LIN {X 0,Y 516.808,Z 520.516,A -85,B 0,C 180,E1 -4959.787,E2 -4959.787} C_VEL
LIN {X 0,Y 517.098,Z 512.267,A -85,B 0,C 180,E1 -4960.969,E2 -4960.969} C_VEL
LIN {X 0,Y 517.442,Z 502.246,A -85,B 0,C 180,E1 -4962.162,E2 -4962.162} C_VEL
LIN {X 0,Y 517.823,Z 491.268,A -85,B 0,C 180,E1 -4963.24,E2 -4963.24} C_VEL
LIN {X 0,Y 518.232,Z 480.256,A -85,B 0,C 180,E1 -4964.129,E2 -4964.129} C_VEL
LIN {X 0,Y 518.655,Z 468.311,A -85,B 0,C 180,E1 -4964.919,E2 -4964.919} C_VEL
LIN {X 0,Y 519.002,Z 455.123,A -85,B 0,C 180,E1 -4965.613,E2 -4965.613} C_VEL
LIN {X 0,Y 519.331,Z 440.839,A -85,B 0,C 180,E1 -4966.176,E2 -4966.176} C_VEL
LIN {X 0,Y 519.289,Z 432.051,A -85,B 0,C 180,E1 -4966.444,E2 -4966.444} C_VEL
LIN {X 0,Y 516.421,Z 418.731,A -85,B 0,C 180,E1 -4966.835,E2 -4966.835} C_VEL
LIN {X 0,Y 516.476,Z 412.491,A -85,B 0,C 180,E1 -4970.128,E2 -4970.128} C_VEL
LIN {X 0,Y 516.541,Z 406.65,A -85,B 0,C 180,E1 -4973.239,E2 -4973.239} C_VEL
LIN {X 0,Y 516.631,Z 401.356,A -85,B 0,C 180,E1 -4976.125,E2 -4976.125} C_VEL
LIN {X 0,Y 516.771,Z 395.647,A -85,B 0,C 180,E1 -4979.314,E2 -4979.314} C_VEL
LIN {X 0,Y 516.843,Z 390.925,A -85,B 0,C 180,E1 -4982.027,E2 -4982.027} C_VEL
LIN {X 0,Y 516.93,Z 386.203,A -85,B 0,C 180,E1 -4984.821,E2 -4984.821} C_VEL
LIN {X 0,Y 517.027,Z 381.474,A -85,B 0,C 180,E1 -4987.712,E2 -4987.712} C_VEL
LIN {X 0,Y 516.923,Z 379.126,A -85,B 0,C 180,E1 -4989.198,E2 -4989.198} C_VEL
LIN {X 0,Y 516.879,Z 378.732,A -85,B 0,C 180,E1 -4989.722,E2 -4989.722} C_VEL
LIN {X 0,Y 516.909,Z 378.724,A -85,B 0,C 180,E1 -4992.761,E2 -4992.761} C_VEL
LIN {X 0,Y 516.926,Z 378.721,A -85,B 0,C 180,E1 -4995.01,E2 -4995.01} C_VEL
LIN {X 0,Y 516.918,Z 378.721,A -85,B 0,C 180,E1 -4998.399,E2 -4998.399} C_VEL
LIN {X 0,Y 516.884,Z 378.727,A -85,B 0,C 180,E1 -5001.284,E2 -5001.284} C_VEL
LIN {X 0,Y 516.894,Z 378.726,A -85,B 0,C 180,E1 -5004.221,E2 -5004.221} C_VEL
LIN {X 0,Y 516.898,Z 378.722,A -85,B 0,C 180,E1 -5007.053,E2 -5007.053} C_VEL
LIN {X 0,Y 516.895,Z 378.722,A -85,B 0,C 180,E1 -5009.796,E2 -5009.796} C_VEL
LIN {X 0,Y 516.931,Z 378.723,A -85,B 0,C 180,E1 -5012.467,E2 -5012.467} C_VEL
LIN {X 0,Y 516.912,Z 378.72,A -85,B 0,C 180,E1 -5015.072,E2 -5015.072} C_VEL
LIN {X 0,Y 516.889,Z 378.723,A -85,B 0,C 180,E1 -5018.462,E2 -5018.462} C_VEL
LIN {X 0,Y 516.905,Z 378.722,A -85,B 0,C 180,E1 -5020.955,E2 -5020.955} C_VEL
LIN {X 0,Y 516.917,Z 378.72,A -85,B 0,C 180,E1 -5023.41,E2 -5023.41} C_VEL
LIN {X 0,Y 516.909,Z 378.721,A -85,B 0,C 180,E1 -5025.834,E2 -5025.834} C_VEL
LIN {X 0,Y 516.954,Z 378.716,A -85,B 0,C 180,E1 -5029.028,E2 -5029.028} C_VEL
LIN {X 0,Y 516.982,Z 378.714,A -85,B 0,C 180,E1 -5032.187,E2 -5032.187} C_VEL
LIN {X 0,Y 517.033,Z 378.704,A -85,B 0,C 180,E1 -5034.54,E2 -5034.54} C_VEL
LIN {X 0,Y 517.086,Z 378.698,A -85,B 0,C 180,E1 -5037.663,E2 -5037.663} C_VEL
LIN {X 0,Y 517.097,Z 378.696,A -85,B 0,C 180,E1 -5040.779,E2 -5040.779} C_VEL
LIN {X 0,Y 517.017,Z 378.71,A -85,B 0,C 180,E1 -5043.117,E2 -5043.117} C_VEL
LIN {X 0,Y 517.013,Z 378.709,A -85,B 0,C 180,E1 -5046.243,E2 -5046.243} C_VEL
LIN {X 0,Y 516.953,Z 378.716,A -85,B 0,C 180,E1 -5049.389,E2 -5049.389} C_VEL
LIN {X 0,Y 516.956,Z 378.715,A -85,B 0,C 180,E1 -5051.807,E2 -5051.807} C_VEL
LIN {X 0,Y 516.951,Z 378.715,A -85,B 0,C 180,E1 -5055.148,E2 -5055.148} C_VEL
LIN {X 0,Y 516.929,Z 378.719,A -85,B 0,C 180,E1 -5058.222,E2 -5058.222} C_VEL
LIN {X 0,Y 516.916,Z 378.721,A -85,B 0,C 180,E1 -5060.701,E2 -5060.701} C_VEL
LIN {X 0,Y 516.915,Z 378.72,A -85,B 0,C 180,E1 -5064.072,E2 -5064.072} C_VEL
LIN {X 0,Y 516.928,Z 378.717,A -85,B 0,C 180,E1 -5066.658,E2 -5066.658} C_VEL
LIN {X 0,Y 516.914,Z 378.72,A -85,B 0,C 180,E1 -5069.524,E2 -5069.524} C_VEL
LIN {X 0,Y 516.898,Z 378.727,A -85,B 0,C 180,E1 -5072.543,E2 -5072.543} C_VEL
LIN {X 0,Y 516.886,Z 378.725,A -85,B 0,C 180,E1 -5075.332,E2 -5075.332} C_VEL
LIN {X 0,Y 516.884,Z 378.725,A -85,B 0,C 180,E1 -5077.943,E2 -5077.943} C_VEL
LIN {X 0,Y 516.907,Z 378.725,A -85,B 0,C 180,E1 -5080.74,E2 -5080.74} C_VEL
LIN {X 0,Y 516.884,Z 378.729,A -85,B 0,C 180,E1 -5083.903,E2 -5083.903} C_VEL
LIN {X 0,Y 516.887,Z 378.729,A -85,B 0,C 180,E1 -5087.169,E2 -5087.169} C_VEL
LIN {X 0,Y 516.955,Z 378.759,A -85,B 0,C 180,E1 -5089.779,E2 -5089.779} C_VEL
LIN {X 0,Y 517.287,Z 382.793,A -85,B 0,C 180,E1 -5091.999,E2 -5091.999} C_VEL
LIN {X 0,Y 517.184,Z 387.817,A -85,B 0,C 180,E1 -5094.621,E2 -5094.621} C_VEL
LIN {X 0,Y 517.022,Z 393.407,A -85,B 0,C 180,E1 -5097.435,E2 -5097.435} C_VEL
LIN {X 0,Y 516.898,Z 399.648,A -85,B 0,C 180,E1 -5100.479,E2 -5100.479} C_VEL
LIN {X 0,Y 516.724,Z 405.675,A -85,B 0,C 180,E1 -5103.331,E2 -5103.331} C_VEL
LIN {X 0,Y 516.658,Z 411.289,A -85,B 0,C 180,E1 -5105.915,E2 -5105.915} C_VEL
LIN {X 0,Y 516.578,Z 416.905,A -85,B 0,C 180,E1 -5108.449,E2 -5108.449} C_VEL
LIN {X 0,Y 516.49,Z 422.509,A -85,B 0,C 180,E1 -5110.939,E2 -5110.939} C_VEL
LIN {X 0,Y 516.463,Z 427.639,A -85,B 0,C 180,E1 -5113.192,E2 -5113.192} C_VEL
LIN {X 0,Y 519.514,Z 442.817,A -85,B 0,C 180,E1 -5113.639,E2 -5113.639} C_VEL
LIN {X 0,Y 519.207,Z 456.026,A -85,B 0,C 180,E1 -5114.065,E2 -5114.065} C_VEL
LIN {X 0,Y 518.82,Z 469.992,A -85,B 0,C 180,E1 -5114.683,E2 -5114.683} C_VEL
LIN {X 0,Y 518.478,Z 482.084,A -85,B 0,C 180,E1 -5115.377,E2 -5115.377} C_VEL
LIN {X 0,Y 518.093,Z 493.307,A -85,B 0,C 180,E1 -5116.167,E2 -5116.167} C_VEL
LIN {X 0,Y 517.657,Z 504.851,A -85,B 0,C 180,E1 -5117.155,E2 -5117.155} C_VEL
LIN {X 0,Y 517.334,Z 515.308,A -85,B 0,C 180,E1 -5118.242,E2 -5118.242} C_VEL
LIN {X 0,Y 517.002,Z 524.755,A -85,B 0,C 180,E1 -5119.425,E2 -5119.425} C_VEL
LIN {X 0,Y 516.71,Z 533.754,A -85,B 0,C 180,E1 -5120.804,E2 -5120.804} C_VEL
LIN {X 0,Y 516.501,Z 541.022,A -85,B 0,C 180,E1 -5122.179,E2 -5122.179} C_VEL
LIN {X 0,Y 516.396,Z 547.553,A -85,B 0,C 180,E1 -5123.749,E2 -5123.749} C_VEL
LIN {X 0,Y 516.306,Z 551.373,A -85,B 0,C 180,E1 -5124.924,E2 -5124.924} C_VEL
LIN {X 0,Y 516.325,Z 554.315,A -85,B 0,C 180,E1 -5126.097,E2 -5126.097} C_VEL
LIN {X 0,Y 516.26,Z 557.002,A -85,B 0,C 180,E1 -5127.659,E2 -5127.659} C_VEL
LIN {X 0,Y 516.157,Z 558.334,A -85,B 0,C 180,E1 -5129.22,E2 -5129.22} C_VEL
LIN {X 0,Y 516.157,Z 558.334,A -85,B 0,C 180,E1 -5130.78,E2 -5130.78} C_VEL
LIN {X 0,Y 516.259,Z 557.005,A -85,B 0,C 180,E1 -5132.341,E2 -5132.341} C_VEL
LIN {X 0,Y 516.325,Z 554.32,A -85,B 0,C 180,E1 -5133.902,E2 -5133.902} C_VEL
LIN {X 0,Y 516.388,Z 550.192,A -85,B 0,C 180,E1 -5135.467,E2 -5135.467} C_VEL
LIN {X 0,Y 516.405,Z 544.503,A -85,B 0,C 180,E1 -5137.035,E2 -5137.035} C_VEL
LIN {X 0,Y 516.599,Z 538.089,A -85,B 0,C 180,E1 -5138.409,E2 -5138.409} C_VEL
LIN {X 0,Y 516.827,Z 530.119,A -85,B 0,C 180,E1 -5139.787,E2 -5139.787} C_VEL
LIN {X 0,Y 517.109,Z 521.781,A -85,B 0,C 180,E1 -5140.969,E2 -5140.969} C_VEL
LIN {X 0,Y 517.458,Z 511.344,A -85,B 0,C 180,E1 -5142.197,E2 -5142.197} C_VEL
LIN {X 0,Y 517.812,Z 500.543,A -85,B 0,C 180,E1 -5143.24,E2 -5143.24} C_VEL
LIN {X 0,Y 518.256,Z 487.977,A -85,B 0,C 180,E1 -5144.229,E2 -5144.229} C_VEL
LIN {X 0,Y 518.701,Z 475.501,A -85,B 0,C 180,E1 -5145.018,E2 -5145.018} C_VEL
LIN {X 0,Y 519.038,Z 462.675,A -85,B 0,C 180,E1 -5145.662,E2 -5145.662} C_VEL
LIN {X 0,Y 519.367,Z 449.107,A -85,B 0,C 180,E1 -5146.176,E2 -5146.176} C_VEL
LIN {X 0,Y 519.32,Z 441.383,A -85,B 0,C 180,E1 -5146.407,E2 -5146.407} C_VEL
LIN {X 0,Y 516.463,Z 427.607,A -85,B 0,C 180,E1 -5146.808,E2 -5146.808} C_VEL
LIN {X 0,Y 516.572,Z 419.95,A -85,B 0,C 180,E1 -5150.157,E2 -5150.157} C_VEL
LIN {X 0,Y 516.615,Z 413.124,A -85,B 0,C 180,E1 -5153.236,E2 -5153.236} C_VEL
LIN {X 0,Y 516.725,Z 406.793,A -85,B 0,C 180,E1 -5156.147,E2 -5156.147} C_VEL
LIN {X 0,Y 516.814,Z 401.952,A -85,B 0,C 180,E1 -5158.421,E2 -5158.421} C_VEL
LIN {X 0,Y 516.969,Z 396.377,A -85,B 0,C 180,E1 -5161.104,E2 -5161.104} C_VEL
LIN {X 0,Y 517.109,Z 390.531,A -85,B 0,C 180,E1 -5163.999,E2 -5163.999} C_VEL
LIN {X 0,Y 517.263,Z 385.229,A -85,B 0,C 180,E1 -5166.714,E2 -5166.714} C_VEL
LIN {X 0,Y 517.184,Z 380.519,A -85,B 0,C 180,E1 -5169.234,E2 -5169.234} C_VEL
LIN {X 0,Y 516.936,Z 378.724,A -85,B 0,C 180,E1 -5170.351,E2 -5170.351} C_VEL
LIN {X 0,Y 516.886,Z 378.728,A -85,B 0,C 180,E1 -5172.831,E2 -5172.831} C_VEL
LIN {X 0,Y 516.883,Z 378.729,A -85,B 0,C 180,E1 -5176.097,E2 -5176.097} C_VEL
LIN {X 0,Y 516.906,Z 378.725,A -85,B 0,C 180,E1 -5179.26,E2 -5179.26} C_VEL
LIN {X 0,Y 516.887,Z 378.723,A -85,B 0,C 180,E1 -5182.056,E2 -5182.056} C_VEL
LIN {X 0,Y 516.897,Z 378.722,A -85,B 0,C 180,E1 -5185.176,E2 -5185.176} C_VEL
LIN {X 0,Y 516.878,Z 378.726,A -85,B 0,C 180,E1 -5187.975,E2 -5187.975} C_VEL
LIN {X 0,Y 516.923,Z 378.723,A -85,B 0,C 180,E1 -5190.696,E2 -5190.696} C_VEL
LIN {X 0,Y 516.944,Z 378.719,A -85,B 0,C 180,E1 -5193.804,E2 -5193.804} C_VEL
LIN {X 0,Y 516.867,Z 378.726,A -85,B 0,C 180,E1 -5196.776,E2 -5196.776} C_VEL
LIN {X 0,Y 516.941,Z 378.716,A -85,B 0,C 180,E1 -5199.732,E2 -5199.732} C_VEL
LIN {X 0,Y 516.931,Z 378.718,A -85,B 0,C 180,E1 -5202.596,E2 -5202.596} C_VEL
LIN {X 0,Y 516.953,Z 378.716,A -85,B 0,C 180,E1 -5205.03,E2 -5205.03} C_VEL
LIN {X 0,Y 516.968,Z 378.714,A -85,B 0,C 180,E1 -5208.234,E2 -5208.234} C_VEL
LIN {X 0,Y 516.971,Z 378.713,A -85,B 0,C 180,E1 -5211.4,E2 -5211.4} C_VEL
LIN {X 0,Y 517.012,Z 378.71,A -85,B 0,C 180,E1 -5213.757,E2 -5213.757} C_VEL
LIN {X 0,Y 517.086,Z 378.698,A -85,B 0,C 180,E1 -5217.663,E2 -5217.663} C_VEL
LIN {X 0,Y 517.096,Z 378.696,A -85,B 0,C 180,E1 -5220.779,E2 -5220.779} C_VEL
LIN {X 0,Y 517.015,Z 378.711,A -85,B 0,C 180,E1 -5223.117,E2 -5223.117} C_VEL
LIN {X 0,Y 517.012,Z 378.71,A -85,B 0,C 180,E1 -5226.243,E2 -5226.243} C_VEL
LIN {X 0,Y 516.954,Z 378.716,A -85,B 0,C 180,E1 -5229.389,E2 -5229.389} C_VEL
LIN {X 0,Y 516.954,Z 378.715,A -85,B 0,C 180,E1 -5231.807,E2 -5231.807} C_VEL
LIN {X 0,Y 516.95,Z 378.715,A -85,B 0,C 180,E1 -5235.148,E2 -5235.148} C_VEL
LIN {X 0,Y 516.928,Z 378.719,A -85,B 0,C 180,E1 -5238.222,E2 -5238.222} C_VEL
LIN {X 0,Y 516.915,Z 378.721,A -85,B 0,C 180,E1 -5240.701,E2 -5240.701} C_VEL
LIN {X 0,Y 516.914,Z 378.722,A -85,B 0,C 180,E1 -5244.072,E2 -5244.072} C_VEL
LIN {X 0,Y 516.928,Z 378.717,A -85,B 0,C 180,E1 -5246.658,E2 -5246.658} C_VEL
LIN {X 0,Y 516.913,Z 378.721,A -85,B 0,C 180,E1 -5249.524,E2 -5249.524} C_VEL
LIN {X 0,Y 516.898,Z 378.726,A -85,B 0,C 180,E1 -5252.543,E2 -5252.543} C_VEL
LIN {X 0,Y 516.886,Z 378.725,A -85,B 0,C 180,E1 -5255.333,E2 -5255.333} C_VEL
LIN {X 0,Y 516.887,Z 378.722,A -85,B 0,C 180,E1 -5257.944,E2 -5257.944} C_VEL
LIN {X 0,Y 516.887,Z 378.727,A -85,B 0,C 180,E1 -5260.741,E2 -5260.741} C_VEL
LIN {X 0,Y 516.886,Z 378.724,A -85,B 0,C 180,E1 -5262.831,E2 -5262.831} C_VEL
LIN {X 0,Y 516.925,Z 378.72,A -85,B 0,C 180,E1 -5265.01,E2 -5265.01} C_VEL
LIN {X 0,Y 516.92,Z 378.722,A -85,B 0,C 180,E1 -5268.398,E2 -5268.398} C_VEL
LIN {X 0,Y 516.869,Z 378.743,A -85,B 0,C 180,E1 -5270.303,E2 -5270.303} C_VEL
LIN {X 0,Y 516.232,Z 379.398,A -85,B 0,C 180,E1 -5270.949,E2 -5270.949} C_VEL
LIN {X 0,Y 513.459,Z 381.35,A -85,B 0,C 180,E1 -5271.988,E2 -5271.988} C_VEL
LIN {X 0,Y 511.089,Z 383.022,A -85,B 0,C 180,E1 -5272.82,E2 -5272.82} C_VEL
LIN {X 0,Y 510.047,Z 384.192,A -85,B 0,C 180,E1 -5273.464,E2 -5273.464} C_VEL
LIN {X 0,Y 509.95,Z 384.556,A -85,B 0,C 180,E1 -5273.682,E2 -5273.682} C_VEL
LIN {X 0,Y 509.869,Z 389.232,A -85,B 0,C 180,E1 -5276.54,E2 -5276.54} C_VEL
LIN {X 0,Y 509.747,Z 393.955,A -85,B 0,C 180,E1 -5279.328,E2 -5279.328} C_VEL
LIN {X 0,Y 509.631,Z 398.68,A -85,B 0,C 180,E1 -5282.039,E2 -5282.039} C_VEL
LIN {X 0,Y 509.537,Z 403.392,A -85,B 0,C 180,E1 -5284.686,E2 -5284.686} C_VEL
LIN {X 0,Y 509.476,Z 408.613,A -85,B 0,C 180,E1 -5287.554,E2 -5287.554} C_VEL
LIN {X 0,Y 509.339,Z 414.363,A -85,B 0,C 180,E1 -5290.661,E2 -5290.661} C_VEL
LIN {X 0,Y 509.343,Z 418.805,A -85,B 0,C 180,E1 -5293.027,E2 -5293.027} C_VEL
LIN {X 0,Y 512.636,Z 433.906,A -85,B 0,C 180,E1 -5293.477,E2 -5293.477} C_VEL
LIN {X 0,Y 512.426,Z 446.731,A -85,B 0,C 180,E1 -5293.907,E2 -5293.907} C_VEL
LIN {X 0,Y 512.057,Z 459.474,A -85,B 0,C 180,E1 -5294.476,E2 -5294.476} C_VEL
LIN {X 0,Y 511.653,Z 471.727,A -85,B 0,C 180,E1 -5295.177,E2 -5295.177} C_VEL
LIN {X 0,Y 511.216,Z 483.048,A -85,B 0,C 180,E1 -5295.978,E2 -5295.978} C_VEL
LIN {X 0,Y 510.749,Z 494.653,A -85,B 0,C 180,E1 -5296.978,E2 -5296.978} C_VEL
LIN {X 0,Y 510.302,Z 505.157,A -85,B 0,C 180,E1 -5298.078,E2 -5298.078} C_VEL
LIN {X 0,Y 510.018,Z 514.633,A -85,B 0,C 180,E1 -5299.279,E2 -5299.279} C_VEL
LIN {X 0,Y 509.69,Z 523.679,A -85,B 0,C 180,E1 -5300.676,E2 -5300.676} C_VEL
LIN {X 0,Y 509.457,Z 530.96,A -85,B 0,C 180,E1 -5302.071,E2 -5302.071} C_VEL
LIN {X 0,Y 509.308,Z 537.501,A -85,B 0,C 180,E1 -5303.662,E2 -5303.662} C_VEL
LIN {X 0,Y 509.239,Z 541.346,A -85,B 0,C 180,E1 -5304.853,E2 -5304.853} C_VEL
LIN {X 0,Y 509.235,Z 544.295,A -85,B 0,C 180,E1 -5306.043,E2 -5306.043} C_VEL
LIN {X 0,Y 509.189,Z 547.011,A -85,B 0,C 180,E1 -5307.627,E2 -5307.627} C_VEL
LIN {X 0,Y 509.07,Z 548.377,A -85,B 0,C 180,E1 -5309.209,E2 -5309.209} C_VEL
LIN {X 0,Y 509.071,Z 548.419,A -85,B 0,C 180,E1 -5310.791,E2 -5310.791} C_VEL
LIN {X 0,Y 509.188,Z 547.134,A -85,B 0,C 180,E1 -5312.373,E2 -5312.373} C_VEL
LIN {X 0,Y 509.235,Z 544.493,A -85,B 0,C 180,E1 -5313.957,E2 -5313.957} C_VEL
LIN {X 0,Y 509.314,Z 540.427,A -85,B 0,C 180,E1 -5315.543,E2 -5315.543} C_VEL
LIN {X 0,Y 509.356,Z 534.811,A -85,B 0,C 180,E1 -5317.134,E2 -5317.134} C_VEL
LIN {X 0,Y 509.548,Z 528.468,A -85,B 0,C 180,E1 -5318.527,E2 -5318.527} C_VEL
LIN {X 0,Y 509.773,Z 520.582,A -85,B 0,C 180,E1 -5319.924,E2 -5319.924} C_VEL
LIN {X 0,Y 510.103,Z 512.332,A -85,B 0,C 180,E1 -5321.121,E2 -5321.121} C_VEL
LIN {X 0,Y 510.453,Z 502.664,A -85,B 0,C 180,E1 -5322.291,E2 -5322.291} C_VEL
LIN {X 0,Y 510.905,Z 491.33,A -85,B 0,C 180,E1 -5323.423,E2 -5323.423} C_VEL
LIN {X 0,Y 511.323,Z 480.317,A -85,B 0,C 180,E1 -5324.324,E2 -5324.324} C_VEL
LIN {X 0,Y 511.776,Z 468.369,A -85,B 0,C 180,E1 -5325.125,E2 -5325.125} C_VEL
LIN {X 0,Y 512.163,Z 455.177,A -85,B 0,C 180,E1 -5325.827,E2 -5325.827} C_VEL
LIN {X 0,Y 512.504,Z 441.427,A -85,B 0,C 180,E1 -5326.38,E2 -5326.38} C_VEL
LIN {X 0,Y 512.552,Z 433.522,A -85,B 0,C 180,E1 -5326.626,E2 -5326.626} C_VEL
LIN {X 0,Y 509.338,Z 418.801,A -85,B 0,C 180,E1 -5327.077,E2 -5327.077} C_VEL
LIN {X 0,Y 509.419,Z 412.833,A -85,B 0,C 180,E1 -5330.259,E2 -5330.259} C_VEL
LIN {X 0,Y 509.465,Z 408.266,A -85,B 0,C 180,E1 -5332.722,E2 -5332.722} C_VEL
LIN {X 0,Y 509.538,Z 403.554,A -85,B 0,C 180,E1 -5335.314,E2 -5335.314} C_VEL
LIN {X 0,Y 509.63,Z 398.693,A -85,B 0,C 180,E1 -5338.044,E2 -5338.044} C_VEL
LIN {X 0,Y 509.747,Z 394.111,A -85,B 0,C 180,E1 -5340.672,E2 -5340.672} C_VEL
LIN {X 0,Y 509.862,Z 389.385,A -85,B 0,C 180,E1 -5343.461,E2 -5343.461} C_VEL
LIN {X 0,Y 509.95,Z 384.66,A -85,B 0,C 180,E1 -5346.343,E2 -5346.343} C_VEL
LIN {X 0,Y 509.954,Z 381.496,A -85,B 0,C 180,E1 -5348.329,E2 -5348.329} C_VEL
LIN {X 0,Y 509.843,Z 379.737,A -85,B 0,C 180,E1 -5349.471,E2 -5349.471} C_VEL
LIN {X 0,Y 509.85,Z 379.601,A -85,B 0,C 180,E1 -5352.488,E2 -5352.488} C_VEL
LIN {X 0,Y 509.86,Z 379.599,A -85,B 0,C 180,E1 -5355.332,E2 -5355.332} C_VEL
LIN {X 0,Y 509.86,Z 379.6,A -85,B 0,C 180,E1 -5358.575,E2 -5358.575} C_VEL
LIN {X 0,Y 509.854,Z 379.599,A -85,B 0,C 180,E1 -5361.786,E2 -5361.786} C_VEL
LIN {X 0,Y 509.85,Z 379.602,A -85,B 0,C 180,E1 -5364.623,E2 -5364.623} C_VEL
LIN {X 0,Y 509.864,Z 379.602,A -85,B 0,C 180,E1 -5367.481,E2 -5367.481} C_VEL
LIN {X 0,Y 509.862,Z 379.598,A -85,B 0,C 180,E1 -5370.274,E2 -5370.274} C_VEL
LIN {X 0,Y 509.888,Z 379.596,A -85,B 0,C 180,E1 -5372.944,E2 -5372.944} C_VEL
LIN {X 0,Y 509.868,Z 379.601,A -85,B 0,C 180,E1 -5375.574,E2 -5375.574} C_VEL
LIN {X 0,Y 509.854,Z 379.602,A -85,B 0,C 180,E1 -5378.998,E2 -5378.998} C_VEL
LIN {X 0,Y 509.885,Z 379.598,A -85,B 0,C 180,E1 -5382.001,E2 -5382.001} C_VEL
LIN {X 0,Y 509.914,Z 379.591,A -85,B 0,C 180,E1 -5384.819,E2 -5384.819} C_VEL
LIN {X 0,Y 509.904,Z 379.593,A -85,B 0,C 180,E1 -5388.124,E2 -5388.124} C_VEL
LIN {X 0,Y 509.918,Z 379.59,A -85,B 0,C 180,E1 -5391.28,E2 -5391.28} C_VEL
LIN {X 0,Y 509.982,Z 379.587,A -85,B 0,C 180,E1 -5393.67,E2 -5393.67} C_VEL
LIN {X 0,Y 510.057,Z 379.573,A -85,B 0,C 180,E1 -5397.631,E2 -5397.631} C_VEL
LIN {X 0,Y 510.067,Z 379.571,A -85,B 0,C 180,E1 -5400.789,E2 -5400.789} C_VEL
LIN {X 0,Y 509.959,Z 379.59,A -85,B 0,C 180,E1 -5403.16,E2 -5403.16} C_VEL
LIN {X 0,Y 509.981,Z 379.586,A -85,B 0,C 180,E1 -5406.33,E2 -5406.33} C_VEL
LIN {X 0,Y 509.915,Z 379.591,A -85,B 0,C 180,E1 -5408.72,E2 -5408.72} C_VEL
LIN {X 0,Y 509.908,Z 379.592,A -85,B 0,C 180,E1 -5411.932,E2 -5411.932} C_VEL
LIN {X 0,Y 509.897,Z 379.594,A -85,B 0,C 180,E1 -5415.242,E2 -5415.242} C_VEL
LIN {X 0,Y 509.892,Z 379.598,A -85,B 0,C 180,E1 -5418.001,E2 -5418.001} C_VEL
LIN {X 0,Y 509.854,Z 379.604,A -85,B 0,C 180,E1 -5421.002,E2 -5421.002} C_VEL
LIN {X 0,Y 509.84,Z 379.599,A -85,B 0,C 180,E1 -5423.563,E2 -5423.563} C_VEL
LIN {X 0,Y 509.914,Z 379.592,A -85,B 0,C 180,E1 -5426.378,E2 -5426.378} C_VEL
LIN {X 0,Y 509.879,Z 379.597,A -85,B 0,C 180,E1 -5428.844,E2 -5428.844} C_VEL
LIN {X 0,Y 509.822,Z 379.603,A -85,B 0,C 180,E1 -5431.59,E2 -5431.59} C_VEL
LIN {X 0,Y 509.857,Z 379.601,A -85,B 0,C 180,E1 -5434.413,E2 -5434.413} C_VEL
LIN {X 0,Y 509.822,Z 379.61,A -85,B 0,C 180,E1 -5437.34,E2 -5437.34} C_VEL
LIN {X 0,Y 509.864,Z 379.603,A -85,B 0,C 180,E1 -5440.38,E2 -5440.38} C_VEL
LIN {X 0,Y 509.825,Z 379.604,A -85,B 0,C 180,E1 -5443.062,E2 -5443.062} C_VEL
LIN {X 0,Y 509.825,Z 379.606,A -85,B 0,C 180,E1 -5445.793,E2 -5445.793} C_VEL
LIN {X 0,Y 509.864,Z 379.603,A -85,B 0,C 180,E1 -5448.575,E2 -5448.575} C_VEL
LIN {X 0,Y 509.913,Z 379.659,A -85,B 0,C 180,E1 -5449.625,E2 -5449.625} C_VEL
LIN {X 0,Y 510.253,Z 383.408,A -85,B 0,C 180,E1 -5451.729,E2 -5451.729} C_VEL
LIN {X 0,Y 510.177,Z 388.375,A -85,B 0,C 180,E1 -5454.367,E2 -5454.367} C_VEL
LIN {X 0,Y 509.979,Z 394.483,A -85,B 0,C 180,E1 -5457.489,E2 -5457.489} C_VEL
LIN {X 0,Y 509.858,Z 400.107,A -85,B 0,C 180,E1 -5460.274,E2 -5460.274} C_VEL
LIN {X 0,Y 509.703,Z 405.632,A -85,B 0,C 180,E1 -5462.934,E2 -5462.934} C_VEL
LIN {X 0,Y 509.618,Z 411.219,A -85,B 0,C 180,E1 -5465.561,E2 -5465.561} C_VEL
LIN {X 0,Y 509.535,Z 416.831,A -85,B 0,C 180,E1 -5468.136,E2 -5468.136} C_VEL
LIN {X 0,Y 509.418,Z 422.437,A -85,B 0,C 180,E1 -5470.664,E2 -5470.664} C_VEL
LIN {X 0,Y 509.369,Z 427.567,A -85,B 0,C 180,E1 -5472.95,E2 -5472.95} C_VEL
LIN {X 0,Y 512.686,Z 443.983,A -85,B 0,C 180,E1 -5473.449,E2 -5473.449} C_VEL
LIN {X 0,Y 512.373,Z 456.977,A -85,B 0,C 180,E1 -5473.887,E2 -5473.887} C_VEL
LIN {X 0,Y 511.967,Z 469.923,A -85,B 0,C 180,E1 -5474.473,E2 -5474.473} C_VEL
LIN {X 0,Y 511.598,Z 482.015,A -85,B 0,C 180,E1 -5475.175,E2 -5475.175} C_VEL
LIN {X 0,Y 511.141,Z 493.238,A -85,B 0,C 180,E1 -5475.975,E2 -5475.975} C_VEL
LIN {X 0,Y 510.703,Z 504.781,A -85,B 0,C 180,E1 -5476.977,E2 -5476.977} C_VEL
LIN {X 0,Y 510.34,Z 515.239,A -85,B 0,C 180,E1 -5478.079,E2 -5478.079} C_VEL
LIN {X 0,Y 509.991,Z 524.686,A -85,B 0,C 180,E1 -5479.278,E2 -5479.278} C_VEL
LIN {X 0,Y 509.673,Z 533.685,A -85,B 0,C 180,E1 -5480.676,E2 -5480.676} C_VEL
LIN {X 0,Y 509.45,Z 540.953,A -85,B 0,C 180,E1 -5482.071,E2 -5482.071} C_VEL
LIN {X 0,Y 509.311,Z 547.484,A -85,B 0,C 180,E1 -5483.662,E2 -5483.662} C_VEL
LIN {X 0,Y 509.239,Z 551.304,A -85,B 0,C 180,E1 -5484.853,E2 -5484.853} C_VEL
LIN {X 0,Y 509.218,Z 554.248,A -85,B 0,C 180,E1 -5486.043,E2 -5486.043} C_VEL
LIN {X 0,Y 509.159,Z 556.942,A -85,B 0,C 180,E1 -5487.627,E2 -5487.627} C_VEL
LIN {X 0,Y 509.071,Z 558.276,A -85,B 0,C 180,E1 -5489.209,E2 -5489.209} C_VEL
LIN {X 0,Y 509.071,Z 558.277,A -85,B 0,C 180,E1 -5490.791,E2 -5490.791} C_VEL
LIN {X 0,Y 509.159,Z 556.945,A -85,B 0,C 180,E1 -5492.373,E2 -5492.373} C_VEL
LIN {X 0,Y 509.218,Z 554.252,A -85,B 0,C 180,E1 -5493.957,E2 -5493.957} C_VEL
LIN {X 0,Y 509.3,Z 550.123,A -85,B 0,C 180,E1 -5495.543,E2 -5495.543} C_VEL
LIN {X 0,Y 509.329,Z 544.433,A -85,B 0,C 180,E1 -5497.134,E2 -5497.134} C_VEL
LIN {X 0,Y 509.553,Z 538.02,A -85,B 0,C 180,E1 -5498.527,E2 -5498.527} C_VEL
LIN {X 0,Y 509.762,Z 530.049,A -85,B 0,C 180,E1 -5499.924,E2 -5499.924} C_VEL
LIN {X 0,Y 510.114,Z 521.712,A -85,B 0,C 180,E1 -5501.121,E2 -5501.121} C_VEL
LIN {X 0,Y 510.461,Z 511.623,A -85,B 0,C 180,E1 -5502.327,E2 -5502.327} C_VEL
LIN {X 0,Y 510.851,Z 500.474,A -85,B 0,C 180,E1 -5503.424,E2 -5503.424} C_VEL
LIN {X 0,Y 511.359,Z 487.908,A -85,B 0,C 180,E1 -5504.425,E2 -5504.425} C_VEL
LIN {X 0,Y 511.825,Z 475.432,A -85,B 0,C 180,E1 -5505.225,E2 -5505.225} C_VEL
LIN {X 0,Y 512.201,Z 462.606,A -85,B 0,C 180,E1 -5505.877,E2 -5505.877} C_VEL
LIN {X 0,Y 512.536,Z 449.63,A -85,B 0,C 180,E1 -5506.378,E2 -5506.378} C_VEL
LIN {X 0,Y 512.455,Z 442.342,A -85,B 0,C 180,E1 -5506.604,E2 -5506.604} C_VEL
LIN {X 0,Y 509.368,Z 427.535,A -85,B 0,C 180,E1 -5507.049,E2 -5507.049} C_VEL
LIN {X 0,Y 509.51,Z 420.264,A -85,B 0,C 180,E1 -5510.287,E2 -5510.287} C_VEL
LIN {X 0,Y 509.544,Z 414.94,A -85,B 0,C 180,E1 -5512.718,E2 -5512.718} C_VEL
LIN {X 0,Y 509.604,Z 409.355,A -85,B 0,C 180,E1 -5515.31,E2 -5515.31} C_VEL
LIN {X 0,Y 509.742,Z 403.535,A -85,B 0,C 180,E1 -5518.068,E2 -5518.068} C_VEL
LIN {X 0,Y 509.888,Z 398.195,A -85,B 0,C 180,E1 -5520.663,E2 -5520.663} C_VEL
LIN {X 0,Y 510.047,Z 392.621,A -85,B 0,C 180,E1 -5523.447,E2 -5523.447} C_VEL
LIN {X 0,Y 510.206,Z 387.051,A -85,B 0,C 180,E1 -5526.322,E2 -5526.322} C_VEL
LIN {X 0,Y 510.249,Z 383.35,A -85,B 0,C 180,E1 -5528.303,E2 -5528.303} C_VEL
LIN {X 0,Y 509.901,Z 379.601,A -85,B 0,C 180,E1 -5530.416,E2 -5530.416} C_VEL
LIN {X 0,Y 509.821,Z 379.605,A -85,B 0,C 180,E1 -5533.572,E2 -5533.572} C_VEL
LIN {X 0,Y 509.82,Z 379.608,A -85,B 0,C 180,E1 -5536.428,E2 -5536.428} C_VEL
LIN {X 0,Y 509.861,Z 379.603,A -85,B 0,C 180,E1 -5539.3,E2 -5539.3} C_VEL
LIN {X 0,Y 509.859,Z 379.599,A -85,B 0,C 180,E1 -5541.785,E2 -5541.785} C_VEL
LIN {X 0,Y 509.848,Z 379.602,A -85,B 0,C 180,E1 -5544.623,E2 -5544.623} C_VEL
LIN {X 0,Y 509.865,Z 379.603,A -85,B 0,C 180,E1 -5547.481,E2 -5547.481} C_VEL
LIN {X 0,Y 509.86,Z 379.599,A -85,B 0,C 180,E1 -5550.274,E2 -5550.274} C_VEL
LIN {X 0,Y 509.886,Z 379.596,A -85,B 0,C 180,E1 -5552.944,E2 -5552.944} C_VEL
LIN {X 0,Y 509.849,Z 379.604,A -85,B 0,C 180,E1 -5555.573,E2 -5555.573} C_VEL
LIN {X 0,Y 509.823,Z 379.602,A -85,B 0,C 180,E1 -5558.149,E2 -5558.149} C_VEL
LIN {X 0,Y 509.867,Z 379.601,A -85,B 0,C 180,E1 -5560.682,E2 -5560.682} C_VEL
LIN {X 0,Y 509.887,Z 379.595,A -85,B 0,C 180,E1 -5563.175,E2 -5563.175} C_VEL
LIN {X 0,Y 509.876,Z 379.599,A -85,B 0,C 180,E1 -5565.634,E2 -5565.634} C_VEL
LIN {X 0,Y 509.916,Z 379.593,A -85,B 0,C 180,E1 -5568.875,E2 -5568.875} C_VEL
LIN {X 0,Y 509.954,Z 379.588,A -85,B 0,C 180,E1 -5572.079,E2 -5572.079} C_VEL
LIN {X 0,Y 509.984,Z 379.582,A -85,B 0,C 180,E1 -5574.464,E2 -5574.464} C_VEL
LIN {X 0,Y 510.057,Z 379.573,A -85,B 0,C 180,E1 -5577.631,E2 -5577.631} C_VEL
LIN {X 0,Y 510.066,Z 379.572,A -85,B 0,C 180,E1 -5580.79,E2 -5580.79} C_VEL
LIN {X 0,Y 509.957,Z 379.59,A -85,B 0,C 180,E1 -5583.16,E2 -5583.16} C_VEL
LIN {X 0,Y 509.981,Z 379.587,A -85,B 0,C 180,E1 -5586.33,E2 -5586.33} C_VEL
LIN {X 0,Y 509.917,Z 379.591,A -85,B 0,C 180,E1 -5588.72,E2 -5588.72} C_VEL
LIN {X 0,Y 509.907,Z 379.592,A -85,B 0,C 180,E1 -5591.932,E2 -5591.932} C_VEL
LIN {X 0,Y 509.896,Z 379.594,A -85,B 0,C 180,E1 -5595.242,E2 -5595.242} C_VEL
LIN {X 0,Y 509.891,Z 379.598,A -85,B 0,C 180,E1 -5598.001,E2 -5598.001} C_VEL
LIN {X 0,Y 509.853,Z 379.604,A -85,B 0,C 180,E1 -5601.002,E2 -5601.002} C_VEL
LIN {X 0,Y 509.839,Z 379.6,A -85,B 0,C 180,E1 -5603.563,E2 -5603.563} C_VEL
LIN {X 0,Y 509.914,Z 379.593,A -85,B 0,C 180,E1 -5606.379,E2 -5606.379} C_VEL
LIN {X 0,Y 509.879,Z 379.597,A -85,B 0,C 180,E1 -5608.844,E2 -5608.844} C_VEL
LIN {X 0,Y 509.822,Z 379.603,A -85,B 0,C 180,E1 -5611.59,E2 -5611.59} C_VEL
LIN {X 0,Y 509.856,Z 379.601,A -85,B 0,C 180,E1 -5614.413,E2 -5614.413} C_VEL
LIN {X 0,Y 509.825,Z 379.608,A -85,B 0,C 180,E1 -5617.34,E2 -5617.34} C_VEL
LIN {X 0,Y 509.841,Z 379.604,A -85,B 0,C 180,E1 -5620.382,E2 -5620.382} C_VEL
LIN {X 0,Y 509.825,Z 379.603,A -85,B 0,C 180,E1 -5623.062,E2 -5623.062} C_VEL
LIN {X 0,Y 509.833,Z 379.604,A -85,B 0,C 180,E1 -5625.792,E2 -5625.792} C_VEL
LIN {X 0,Y 509.861,Z 379.603,A -85,B 0,C 180,E1 -5628.575,E2 -5628.575} C_VEL
LIN {X 0,Y 509.846,Z 379.771,A -85,B 0,C 180,E1 -5630.648,E2 -5630.648} C_VEL
LIN {X 0,Y 510.005,Z 383.546,A -85,B 0,C 180,E1 -5633.059,E2 -5633.059} C_VEL
LIN {X 0,Y 509.95,Z 384.556,A -85,B 0,C 180,E1 -5633.682,E2 -5633.682} C_VEL
LIN {X 0,Y 509.258,Z 385.694,A -85,B 0,C 180,E1 -5634.329,E2 -5634.329} C_VEL
LIN {X 0,Y 506.413,Z 387.769,A -85,B 0,C 180,E1 -5635.374,E2 -5635.374} C_VEL
LIN {X 0,Y 503.999,Z 389.457,A -85,B 0,C 180,E1 -5636.216,E2 -5636.216} C_VEL
LIN {X 0,Y 502.926,Z 390.663,A -85,B 0,C 180,E1 -5636.867,E2 -5636.867} C_VEL
LIN {X 0,Y 502.818,Z 391.041,A -85,B 0,C 180,E1 -5637.088,E2 -5637.088} C_VEL
LIN {X 0,Y 502.68,Z 396.105,A -85,B 0,C 180,E1 -5640.092,E2 -5640.092} C_VEL
LIN {X 0,Y 502.526,Z 402.051,A -85,B 0,C 180,E1 -5643.517,E2 -5643.517} C_VEL
LIN {X 0,Y 502.426,Z 406.581,A -85,B 0,C 180,E1 -5646.068,E2 -5646.068} C_VEL
LIN {X 0,Y 502.352,Z 411.295,A -85,B 0,C 180,E1 -5648.67,E2 -5648.67} C_VEL
LIN {X 0,Y 502.27,Z 415.998,A -85,B 0,C 180,E1 -5651.227,E2 -5651.227} C_VEL
LIN {X 0,Y 502.269,Z 418.904,A -85,B 0,C 180,E1 -5652.781,E2 -5652.781} C_VEL
LIN {X 0,Y 505.53,Z 433.41,A -85,B 0,C 180,E1 -5653.222,E2 -5653.222} C_VEL
LIN {X 0,Y 505.791,Z 437.737,A -85,B 0,C 180,E1 -5653.36,E2 -5653.36} C_VEL
LIN {X 0,Y 505.452,Z 451.008,A -85,B 0,C 180,E1 -5653.854,E2 -5653.854} C_VEL
LIN {X 0,Y 505.087,Z 463.386,A -85,B 0,C 180,E1 -5654.464,E2 -5654.464} C_VEL
LIN {X 0,Y 504.572,Z 476.324,A -85,B 0,C 180,E1 -5655.274,E2 -5655.274} C_VEL
LIN {X 0,Y 504.083,Z 488.048,A -85,B 0,C 180,E1 -5656.187,E2 -5656.187} C_VEL
LIN {X 0,Y 503.621,Z 498.87,A -85,B 0,C 180,E1 -5657.211,E2 -5657.211} C_VEL
LIN {X 0,Y 503.289,Z 508.572,A -85,B 0,C 180,E1 -5658.318,E2 -5658.318} C_VEL
LIN {X 0,Y 502.859,Z 517.465,A -85,B 0,C 180,E1 -5659.532,E2 -5659.532} C_VEL
LIN {X 0,Y 502.569,Z 525.977,A -85,B 0,C 180,E1 -5660.949,E2 -5660.949} C_VEL
LIN {X 0,Y 502.336,Z 532.836,A -85,B 0,C 180,E1 -5662.362,E2 -5662.362} C_VEL
LIN {X 0,Y 502.235,Z 537.572,A -85,B 0,C 180,E1 -5663.572,E2 -5663.572} C_VEL
LIN {X 0,Y 502.175,Z 541.416,A -85,B 0,C 180,E1 -5664.781,E2 -5664.781} C_VEL
LIN {X 0,Y 502.132,Z 544.366,A -85,B 0,C 180,E1 -5665.987,E2 -5665.987} C_VEL
LIN {X 0,Y 502.09,Z 547.081,A -85,B 0,C 180,E1 -5667.593,E2 -5667.593} C_VEL
LIN {X 0,Y 501.987,Z 548.446,A -85,B 0,C 180,E1 -5669.198,E2 -5669.198} C_VEL
LIN {X 0,Y 501.988,Z 548.488,A -85,B 0,C 180,E1 -5670.802,E2 -5670.802} C_VEL
LIN {X 0,Y 502.09,Z 547.202,A -85,B 0,C 180,E1 -5672.407,E2 -5672.407} C_VEL
LIN {X 0,Y 502.132,Z 544.56,A -85,B 0,C 180,E1 -5674.013,E2 -5674.013} C_VEL
LIN {X 0,Y 502.225,Z 540.495,A -85,B 0,C 180,E1 -5675.622,E2 -5675.622} C_VEL
LIN {X 0,Y 502.3,Z 534.877,A -85,B 0,C 180,E1 -5677.234,E2 -5677.234} C_VEL
LIN {X 0,Y 502.507,Z 528.534,A -85,B 0,C 180,E1 -5678.647,E2 -5678.647} C_VEL
LIN {X 0,Y 502.726,Z 520.647,A -85,B 0,C 180,E1 -5680.064,E2 -5680.064} C_VEL
LIN {X 0,Y 503.119,Z 512.396,A -85,B 0,C 180,E1 -5681.278,E2 -5681.278} C_VEL
LIN {X 0,Y 503.493,Z 502.459,A -85,B 0,C 180,E1 -5682.495,E2 -5682.495} C_VEL
LIN {X 0,Y 503.99,Z 491.392,A -85,B 0,C 180,E1 -5683.61,E2 -5683.61} C_VEL
LIN {X 0,Y 504.409,Z 480.378,A -85,B 0,C 180,E1 -5684.525,E2 -5684.525} C_VEL
LIN {X 0,Y 504.902,Z 468.428,A -85,B 0,C 180,E1 -5685.336,E2 -5685.336} C_VEL
LIN {X 0,Y 505.347,Z 455.232,A -85,B 0,C 180,E1 -5686.046,E2 -5686.046} C_VEL
LIN {X 0,Y 505.703,Z 441.391,A -85,B 0,C 180,E1 -5686.609,E2 -5686.609} C_VEL
LIN {X 0,Y 505.736,Z 434.743,A -85,B 0,C 180,E1 -5686.824,E2 -5686.824} C_VEL
LIN {X 0,Y 502.687,Z 421.018,A -85,B 0,C 180,E1 -5687.257,E2 -5687.257} C_VEL
LIN {X 0,Y 502.278,Z 418.872,A -85,B 0,C 180,E1 -5687.324,E2 -5687.324} C_VEL
LIN {X 0,Y 502.338,Z 413.031,A -85,B 0,C 180,E1 -5690.473,E2 -5690.473} C_VEL
LIN {X 0,Y 502.396,Z 408.314,A -85,B 0,C 180,E1 -5693.06,E2 -5693.06} C_VEL
LIN {X 0,Y 502.474,Z 403.603,A -85,B 0,C 180,E1 -5695.696,E2 -5695.696} C_VEL
LIN {X 0,Y 502.579,Z 398.882,A -85,B 0,C 180,E1 -5698.389,E2 -5698.389} C_VEL
LIN {X 0,Y 502.76,Z 393.567,A -85,B 0,C 180,E1 -5701.492,E2 -5701.492} C_VEL
LIN {X 0,Y 502.818,Z 389.422,A -85,B 0,C 180,E1 -5703.993,E2 -5703.993} C_VEL
LIN {X 0,Y 502.97,Z 384.25,A -85,B 0,C 180,E1 -5707.206,E2 -5707.206} C_VEL
LIN {X 0,Y 502.777,Z 380.489,A -85,B 0,C 180,E1 -5709.753,E2 -5709.753} C_VEL
LIN {X 0,Y 502.805,Z 380.478,A -85,B 0,C 180,E1 -5712.199,E2 -5712.199} C_VEL
LIN {X 0,Y 502.804,Z 380.478,A -85,B 0,C 180,E1 -5715.468,E2 -5715.468} C_VEL
LIN {X 0,Y 502.823,Z 380.477,A -85,B 0,C 180,E1 -5718.934,E2 -5718.934} C_VEL
LIN {X 0,Y 502.797,Z 380.478,A -85,B 0,C 180,E1 -5722.046,E2 -5722.046} C_VEL
LIN {X 0,Y 502.813,Z 380.476,A -85,B 0,C 180,E1 -5725.035,E2 -5725.035} C_VEL
LIN {X 0,Y 502.786,Z 380.481,A -85,B 0,C 180,E1 -5727.915,E2 -5727.915} C_VEL
LIN {X 0,Y 502.827,Z 380.478,A -85,B 0,C 180,E1 -5730.712,E2 -5730.712} C_VEL
LIN {X 0,Y 502.866,Z 380.469,A -85,B 0,C 180,E1 -5733.439,E2 -5733.439} C_VEL
LIN {X 0,Y 502.789,Z 380.479,A -85,B 0,C 180,E1 -5736.086,E2 -5736.086} C_VEL
LIN {X 0,Y 502.787,Z 380.482,A -85,B 0,C 180,E1 -5738.689,E2 -5738.689} C_VEL
LIN {X 0,Y 502.833,Z 380.473,A -85,B 0,C 180,E1 -5741.248,E2 -5741.248} C_VEL
LIN {X 0,Y 502.825,Z 380.48,A -85,B 0,C 180,E1 -5743.767,E2 -5743.767} C_VEL
LIN {X 0,Y 502.839,Z 380.472,A -85,B 0,C 180,E1 -5746.255,E2 -5746.255} C_VEL
LIN {X 0,Y 502.88,Z 380.472,A -85,B 0,C 180,E1 -5748.717,E2 -5748.717} C_VEL
LIN {X 0,Y 502.905,Z 380.47,A -85,B 0,C 180,E1 -5751.967,E2 -5751.967} C_VEL
LIN {X 0,Y 502.941,Z 380.46,A -85,B 0,C 180,E1 -5754.386,E2 -5754.386} C_VEL
LIN {X 0,Y 503.027,Z 380.449,A -85,B 0,C 180,E1 -5757.598,E2 -5757.598} C_VEL
LIN {X 0,Y 503.03,Z 380.454,A -85,B 0,C 180,E1 -5760,E2 -5760} C_VEL
LIN {X 0,Y 503.028,Z 380.449,A -85,B 0,C 180,E1 -5762.402,E2 -5762.402} C_VEL
LIN {X 0,Y 502.941,Z 380.459,A -85,B 0,C 180,E1 -5765.613,E2 -5765.613} C_VEL
LIN {X 0,Y 502.904,Z 380.469,A -85,B 0,C 180,E1 -5768.033,E2 -5768.033} C_VEL
LIN {X 0,Y 502.881,Z 380.472,A -85,B 0,C 180,E1 -5771.283,E2 -5771.283} C_VEL
LIN {X 0,Y 502.855,Z 380.476,A -85,B 0,C 180,E1 -5774.57,E2 -5774.57} C_VEL
LIN {X 0,Y 502.865,Z 380.475,A -85,B 0,C 180,E1 -5777.907,E2 -5777.907} C_VEL
LIN {X 0,Y 502.832,Z 380.474,A -85,B 0,C 180,E1 -5780.536,E2 -5780.536} C_VEL
LIN {X 0,Y 502.8,Z 380.478,A -85,B 0,C 180,E1 -5783.04,E2 -5783.04} C_VEL
LIN {X 0,Y 502.843,Z 380.474,A -85,B 0,C 180,E1 -5785.675,E2 -5785.675} C_VEL
LIN {X 0,Y 502.843,Z 380.472,A -85,B 0,C 180,E1 -5788.372,E2 -5788.372} C_VEL
LIN {X 0,Y 502.795,Z 380.478,A -85,B 0,C 180,E1 -5791.499,E2 -5791.499} C_VEL
LIN {X 0,Y 502.809,Z 380.479,A -85,B 0,C 180,E1 -5794.445,E2 -5794.445} C_VEL
LIN {X 0,Y 502.784,Z 380.485,A -85,B 0,C 180,E1 -5797.178,E2 -5797.178} C_VEL
LIN {X 0,Y 502.829,Z 380.476,A -85,B 0,C 180,E1 -5800.011,E2 -5800.011} C_VEL
LIN {X 0,Y 502.774,Z 380.483,A -85,B 0,C 180,E1 -5803.231,E2 -5803.231} C_VEL
LIN {X 0,Y 502.781,Z 380.485,A -85,B 0,C 180,E1 -5805.66,E2 -5805.66} C_VEL
LIN {X 0,Y 502.828,Z 380.479,A -85,B 0,C 180,E1 -5809.004,E2 -5809.004} C_VEL
LIN {X 0,Y 502.859,Z 380.557,A -85,B 0,C 180,E1 -5809.467,E2 -5809.467} C_VEL
LIN {X 0,Y 503.215,Z 384.036,A -85,B 0,C 180,E1 -5811.454,E2 -5811.454} C_VEL
LIN {X 0,Y 503.171,Z 388.928,A -85,B 0,C 180,E1 -5814.107,E2 -5814.107} C_VEL
LIN {X 0,Y 502.972,Z 394.449,A -85,B 0,C 180,E1 -5816.979,E2 -5816.979} C_VEL
LIN {X 0,Y 502.82,Z 400.566,A -85,B 0,C 180,E1 -5820.064,E2 -5820.064} C_VEL
LIN {X 0,Y 502.647,Z 407.586,A -85,B 0,C 180,E1 -5823.489,E2 -5823.489} C_VEL
LIN {X 0,Y 502.493,Z 413.028,A -85,B 0,C 180,E1 -5826.071,E2 -5826.071} C_VEL
LIN {X 0,Y 502.436,Z 418.627,A -85,B 0,C 180,E1 -5828.673,E2 -5828.673} C_VEL
LIN {X 0,Y 502.331,Z 424.231,A -85,B 0,C 180,E1 -5831.229,E2 -5831.229} C_VEL
LIN {X 0,Y 502.331,Z 427.496,A -85,B 0,C 180,E1 -5832.704,E2 -5832.704} C_VEL
LIN {X 0,Y 505.802,Z 444.288,A -85,B 0,C 180,E1 -5833.228,E2 -5833.228} C_VEL
LIN {X 0,Y 505.519,Z 458.024,A -85,B 0,C 180,E1 -5833.707,E2 -5833.707} C_VEL
LIN {X 0,Y 505.078,Z 471.818,A -85,B 0,C 180,E1 -5834.36,E2 -5834.36} C_VEL
LIN {X 0,Y 504.571,Z 484.979,A -85,B 0,C 180,E1 -5835.171,E2 -5835.171} C_VEL
LIN {X 0,Y 504.106,Z 496.881,A -85,B 0,C 180,E1 -5836.084,E2 -5836.084} C_VEL
LIN {X 0,Y 503.612,Z 507.75,A -85,B 0,C 180,E1 -5837.098,E2 -5837.098} C_VEL
LIN {X 0,Y 503.219,Z 518.49,A -85,B 0,C 180,E1 -5838.316,E2 -5838.316} C_VEL
LIN {X 0,Y 502.836,Z 527.356,A -85,B 0,C 180,E1 -5839.531,E2 -5839.531} C_VEL
LIN {X 0,Y 502.554,Z 535.851,A -85,B 0,C 180,E1 -5840.948,E2 -5840.948} C_VEL
LIN {X 0,Y 502.321,Z 542.697,A -85,B 0,C 180,E1 -5842.362,E2 -5842.362} C_VEL
LIN {X 0,Y 502.234,Z 547.414,A -85,B 0,C 180,E1 -5843.572,E2 -5843.572} C_VEL
LIN {X 0,Y 502.172,Z 551.235,A -85,B 0,C 180,E1 -5844.781,E2 -5844.781} C_VEL
LIN {X 0,Y 502.113,Z 554.179,A -85,B 0,C 180,E1 -5845.987,E2 -5845.987} C_VEL
LIN {X 0,Y 502.064,Z 556.873,A -85,B 0,C 180,E1 -5847.593,E2 -5847.593} C_VEL
LIN {X 0,Y 501.988,Z 558.208,A -85,B 0,C 180,E1 -5849.198,E2 -5849.198} C_VEL
LIN {X 0,Y 501.988,Z 558.208,A -85,B 0,C 180,E1 -5850.802,E2 -5850.802} C_VEL
LIN {X 0,Y 502.064,Z 556.876,A -85,B 0,C 180,E1 -5852.407,E2 -5852.407} C_VEL
LIN {X 0,Y 502.113,Z 554.183,A -85,B 0,C 180,E1 -5854.013,E2 -5854.013} C_VEL
LIN {X 0,Y 502.216,Z 550.054,A -85,B 0,C 180,E1 -5855.622,E2 -5855.622} C_VEL
LIN {X 0,Y 502.254,Z 544.364,A -85,B 0,C 180,E1 -5857.235,E2 -5857.235} C_VEL
LIN {X 0,Y 502.482,Z 537.95,A -85,B 0,C 180,E1 -5858.647,E2 -5858.647} C_VEL
LIN {X 0,Y 502.731,Z 529.98,A -85,B 0,C 180,E1 -5860.064,E2 -5860.064} C_VEL
LIN {X 0,Y 503.1,Z 521.643,A -85,B 0,C 180,E1 -5861.278,E2 -5861.278} C_VEL
LIN {X 0,Y 503.513,Z 510.967,A -85,B 0,C 180,E1 -5862.566,E2 -5862.566} C_VEL
LIN {X 0,Y 503.92,Z 500.405,A -85,B 0,C 180,E1 -5863.612,E2 -5863.612} C_VEL
LIN {X 0,Y 504.454,Z 487.839,A -85,B 0,C 180,E1 -5864.626,E2 -5864.626} C_VEL
LIN {X 0,Y 504.952,Z 475.363,A -85,B 0,C 180,E1 -5865.437,E2 -5865.437} C_VEL
LIN {X 0,Y 505.36,Z 462.537,A -85,B 0,C 180,E1 -5866.097,E2 -5866.097} C_VEL
LIN {X 0,Y 505.718,Z 448.814,A -85,B 0,C 180,E1 -5866.631,E2 -5866.631} C_VEL
LIN {X 0,Y 505.574,Z 443.094,A -85,B 0,C 180,E1 -5866.814,E2 -5866.814} C_VEL
LIN {X 0,Y 502.468,Z 428.581,A -85,B 0,C 180,E1 -5867.251,E2 -5867.251} C_VEL
LIN {X 0,Y 502.33,Z 427.464,A -85,B 0,C 180,E1 -5867.296,E2 -5867.296} C_VEL
LIN {X 0,Y 502.428,Z 420.474,A -85,B 0,C 180,E1 -5870.469,E2 -5870.469} C_VEL
LIN {X 0,Y 502.482,Z 414.891,A -85,B 0,C 180,E1 -5873.056,E2 -5873.056} C_VEL
LIN {X 0,Y 502.56,Z 409.302,A -85,B 0,C 180,E1 -5875.691,E2 -5875.691} C_VEL
LIN {X 0,Y 502.7,Z 403.723,A -85,B 0,C 180,E1 -5878.381,E2 -5878.381} C_VEL
LIN {X 0,Y 502.884,Z 398.157,A -85,B 0,C 180,E1 -5881.137,E2 -5881.137} C_VEL
LIN {X 0,Y 503.047,Z 392.589,A -85,B 0,C 180,E1 -5883.975,E2 -5883.975} C_VEL
LIN {X 0,Y 503.226,Z 387.026,A -85,B 0,C 180,E1 -5886.908,E2 -5886.908} C_VEL
LIN {X 0,Y 503.185,Z 383.324,A -85,B 0,C 180,E1 -5888.941,E2 -5888.941} C_VEL
LIN {X 0,Y 502.824,Z 380.482,A -85,B 0,C 180,E1 -5890.668,E2 -5890.668} C_VEL
LIN {X 0,Y 502.773,Z 380.484,A -85,B 0,C 180,E1 -5893.374,E2 -5893.374} C_VEL
LIN {X 0,Y 502.772,Z 380.484,A -85,B 0,C 180,E1 -5896.626,E2 -5896.626} C_VEL
LIN {X 0,Y 502.828,Z 380.477,A -85,B 0,C 180,E1 -5899.004,E2 -5899.004} C_VEL
LIN {X 0,Y 502.8,Z 380.478,A -85,B 0,C 180,E1 -5902.047,E2 -5902.047} C_VEL
LIN {X 0,Y 502.812,Z 380.477,A -85,B 0,C 180,E1 -5905.035,E2 -5905.035} C_VEL
LIN {X 0,Y 502.786,Z 380.482,A -85,B 0,C 180,E1 -5907.916,E2 -5907.916} C_VEL
LIN {X 0,Y 502.826,Z 380.48,A -85,B 0,C 180,E1 -5910.712,E2 -5910.712} C_VEL
LIN {X 0,Y 502.864,Z 380.47,A -85,B 0,C 180,E1 -5913.439,E2 -5913.439} C_VEL
LIN {X 0,Y 502.777,Z 380.482,A -85,B 0,C 180,E1 -5916.086,E2 -5916.086} C_VEL
LIN {X 0,Y 502.785,Z 380.482,A -85,B 0,C 180,E1 -5918.689,E2 -5918.689} C_VEL
LIN {X 0,Y 502.833,Z 380.473,A -85,B 0,C 180,E1 -5921.248,E2 -5921.248} C_VEL
LIN {X 0,Y 502.824,Z 380.48,A -85,B 0,C 180,E1 -5923.767,E2 -5923.767} C_VEL
LIN {X 0,Y 502.838,Z 380.472,A -85,B 0,C 180,E1 -5926.255,E2 -5926.255} C_VEL
LIN {X 0,Y 502.88,Z 380.471,A -85,B 0,C 180,E1 -5928.717,E2 -5928.717} C_VEL
LIN {X 0,Y 502.904,Z 380.468,A -85,B 0,C 180,E1 -5931.967,E2 -5931.967} C_VEL
LIN {X 0,Y 502.94,Z 380.46,A -85,B 0,C 180,E1 -5934.387,E2 -5934.387} C_VEL
LIN {X 0,Y 503.027,Z 380.449,A -85,B 0,C 180,E1 -5937.598,E2 -5937.598} C_VEL
LIN {X 0,Y 503.03,Z 380.454,A -85,B 0,C 180,E1 -5940,E2 -5940} C_VEL
LIN {X 0,Y 503.025,Z 380.449,A -85,B 0,C 180,E1 -5942.402,E2 -5942.402} C_VEL
LIN {X 0,Y 502.94,Z 380.46,A -85,B 0,C 180,E1 -5945.614,E2 -5945.614} C_VEL
LIN {X 0,Y 502.904,Z 380.469,A -85,B 0,C 180,E1 -5948.033,E2 -5948.033} C_VEL
LIN {X 0,Y 502.879,Z 380.472,A -85,B 0,C 180,E1 -5951.283,E2 -5951.283} C_VEL
LIN {X 0,Y 502.854,Z 380.475,A -85,B 0,C 180,E1 -5954.571,E2 -5954.571} C_VEL
LIN {X 0,Y 502.864,Z 380.474,A -85,B 0,C 180,E1 -5957.907,E2 -5957.907} C_VEL
LIN {X 0,Y 502.831,Z 380.474,A -85,B 0,C 180,E1 -5960.536,E2 -5960.536} C_VEL
LIN {X 0,Y 502.799,Z 380.48,A -85,B 0,C 180,E1 -5963.04,E2 -5963.04} C_VEL
LIN {X 0,Y 502.843,Z 380.475,A -85,B 0,C 180,E1 -5965.676,E2 -5965.676} C_VEL
LIN {X 0,Y 502.842,Z 380.472,A -85,B 0,C 180,E1 -5968.373,E2 -5968.373} C_VEL
LIN {X 0,Y 502.795,Z 380.478,A -85,B 0,C 180,E1 -5971.499,E2 -5971.499} C_VEL
LIN {X 0,Y 502.809,Z 380.478,A -85,B 0,C 180,E1 -5974.445,E2 -5974.445} C_VEL
LIN {X 0,Y 502.786,Z 380.484,A -85,B 0,C 180,E1 -5977.179,E2 -5977.179} C_VEL
LIN {X 0,Y 502.79,Z 380.479,A -85,B 0,C 180,E1 -5980.015,E2 -5980.015} C_VEL
LIN {X 0,Y 502.804,Z 380.482,A -85,B 0,C 180,E1 -5982.199,E2 -5982.199} C_VEL
LIN {X 0,Y 502.803,Z 380.482,A -85,B 0,C 180,E1 -5985.468,E2 -5985.468} C_VEL
LIN {X 0,Y 502.832,Z 380.475,A -85,B 0,C 180,E1 -5987.864,E2 -5987.864} C_VEL
LIN {X 0,Y 502.78,Z 380.485,A -85,B 0,C 180,E1 -5990.247,E2 -5990.247} C_VEL
LIN {X 0,Y 502.936,Z 382.961,A -85,B 0,C 180,E1 -5992.059,E2 -5992.059} C_VEL
LIN {X 0,Y 502.9,Z 386.266,A -85,B 0,C 180,E1 -5994.15,E2 -5994.15} C_VEL
LIN {X 0,Y 502.818,Z 391.041,A -85,B 0,C 180,E1 -5997.088,E2 -5997.088} C_VEL
LIN {X 0,Y 502.093,Z 392.217,A -85,B 0,C 180,E1 -5997.743,E2 -5997.743} C_VEL
LIN {X 0,Y 499.196,Z 394.34,A -85,B 0,C 180,E1 -5998.801,E2 -5998.801} C_VEL
LIN {X 0,Y 496.758,Z 396.065,A -85,B 0,C 180,E1 -5999.652,E2 -5999.652} C_VEL
LIN {X 0,Y 495.685,Z 397.301,A -85,B 0,C 180,E1 -6000.312,E2 -6000.312} C_VEL
LIN {X 0,Y 495.581,Z 397.691,A -85,B 0,C 180,E1 -6000.537,E2 -6000.537} C_VEL
LIN {X 0,Y 495.475,Z 402.483,A -85,B 0,C 180,E1 -6003.331,E2 -6003.331} C_VEL
LIN {X 0,Y 495.395,Z 406.635,A -85,B 0,C 180,E1 -6005.706,E2 -6005.706} C_VEL
LIN {X 0,Y 495.3,Z 411.348,A -85,B 0,C 180,E1 -6008.351,E2 -6008.351} C_VEL
LIN {X 0,Y 495.204,Z 416.063,A -85,B 0,C 180,E1 -6010.948,E2 -6010.948} C_VEL
LIN {X 0,Y 495.207,Z 418.94,A -85,B 0,C 180,E1 -6012.521,E2 -6012.521} C_VEL
LIN {X 0,Y 498.671,Z 434.509,A -85,B 0,C 180,E1 -6013.013,E2 -6013.013} C_VEL
LIN {X 0,Y 499.029,Z 436.894,A -85,B 0,C 180,E1 -6013.096,E2 -6013.096} C_VEL
LIN {X 0,Y 498.632,Z 451.091,A -85,B 0,C 180,E1 -6013.627,E2 -6013.627} C_VEL
LIN {X 0,Y 498.248,Z 463.466,A -85,B 0,C 180,E1 -6014.245,E2 -6014.245} C_VEL
LIN {X 0,Y 497.704,Z 476.402,A -85,B 0,C 180,E1 -6015.066,E2 -6015.066} C_VEL
LIN {X 0,Y 497.177,Z 488.125,A -85,B 0,C 180,E1 -6015.991,E2 -6015.991} C_VEL
LIN {X 0,Y 496.667,Z 498.946,A -85,B 0,C 180,E1 -6017.029,E2 -6017.029} C_VEL
LIN {X 0,Y 496.279,Z 508.889,A -85,B 0,C 180,E1 -6018.182,E2 -6018.182} C_VEL
LIN {X 0,Y 495.855,Z 517.538,A -85,B 0,C 180,E1 -6019.382,E2 -6019.382} C_VEL
LIN {X 0,Y 495.541,Z 526.05,A -85,B 0,C 180,E1 -6020.819,E2 -6020.819} C_VEL
LIN {X 0,Y 495.274,Z 532.908,A -85,B 0,C 180,E1 -6022.253,E2 -6022.253} C_VEL
LIN {X 0,Y 495.147,Z 538.559,A -85,B 0,C 180,E1 -6023.744,E2 -6023.744} C_VEL
LIN {X 0,Y 495.032,Z 542.549,A -85,B 0,C 180,E1 -6025.114,E2 -6025.114} C_VEL
LIN {X 0,Y 495.036,Z 545.966,A -85,B 0,C 180,E1 -6026.745,E2 -6026.745} C_VEL
LIN {X 0,Y 494.961,Z 547.998,A -85,B 0,C 180,E1 -6028.373,E2 -6028.373} C_VEL
LIN {X 0,Y 494.897,Z 548.701,A -85,B 0,C 180,E1 -6030,E2 -6030} C_VEL
LIN {X 0,Y 494.96,Z 548.08,A -85,B 0,C 180,E1 -6031.627,E2 -6031.627} C_VEL
LIN {X 0,Y 495.035,Z 546.121,A -85,B 0,C 180,E1 -6033.256,E2 -6033.256} C_VEL
LIN {X 0,Y 495.031,Z 542.78,A -85,B 0,C 180,E1 -6034.887,E2 -6034.887} C_VEL
LIN {X 0,Y 495.143,Z 538.887,A -85,B 0,C 180,E1 -6036.252,E2 -6036.252} C_VEL
LIN {X 0,Y 495.27,Z 533.305,A -85,B 0,C 180,E1 -6037.748,E2 -6037.748} C_VEL
LIN {X 0,Y 495.536,Z 526.535,A -85,B 0,C 180,E1 -6039.181,E2 -6039.181} C_VEL
LIN {X 0,Y 495.829,Z 518.126,A -85,B 0,C 180,E1 -6040.618,E2 -6040.618} C_VEL
LIN {X 0,Y 496.302,Z 508.406,A -85,B 0,C 180,E1 -6041.97,E2 -6041.97} C_VEL
LIN {X 0,Y 496.678,Z 498.716,A -85,B 0,C 180,E1 -6043.085,E2 -6043.085} C_VEL
LIN {X 0,Y 497.2,Z 487.962,A -85,B 0,C 180,E1 -6044.113,E2 -6044.113} C_VEL
LIN {X 0,Y 497.719,Z 476.196,A -85,B 0,C 180,E1 -6045.038,E2 -6045.038} C_VEL
LIN {X 0,Y 498.244,Z 463.214,A -85,B 0,C 180,E1 -6045.861,E2 -6045.861} C_VEL
LIN {X 0,Y 498.684,Z 450.181,A -85,B 0,C 180,E1 -6046.504,E2 -6046.504} C_VEL
LIN {X 0,Y 498.924,Z 435.895,A -85,B 0,C 180,E1 -6047.029,E2 -6047.029} C_VEL
LIN {X 0,Y 495.828,Z 421.862,A -85,B 0,C 180,E1 -6047.489,E2 -6047.489} C_VEL
LIN {X 0,Y 495.212,Z 418.926,A -85,B 0,C 180,E1 -6047.583,E2 -6047.583} C_VEL
LIN {X 0,Y 495.253,Z 413.081,A -85,B 0,C 180,E1 -6050.779,E2 -6050.779} C_VEL
LIN {X 0,Y 495.327,Z 408.369,A -85,B 0,C 180,E1 -6053.408,E2 -6053.408} C_VEL
LIN {X 0,Y 495.427,Z 403.655,A -85,B 0,C 180,E1 -6056.089,E2 -6056.089} C_VEL
LIN {X 0,Y 495.542,Z 398.926,A -85,B 0,C 180,E1 -6058.83,E2 -6058.83} C_VEL
LIN {X 0,Y 495.727,Z 394.054,A -85,B 0,C 180,E1 -6061.72,E2 -6061.72} C_VEL
LIN {X 0,Y 495.805,Z 389.197,A -85,B 0,C 180,E1 -6064.7,E2 -6064.7} C_VEL
LIN {X 0,Y 495.915,Z 384.722,A -85,B 0,C 180,E1 -6067.545,E2 -6067.545} C_VEL
LIN {X 0,Y 495.754,Z 381.555,A -85,B 0,C 180,E1 -6069.638,E2 -6069.638} C_VEL
LIN {X 0,Y 495.78,Z 381.356,A -85,B 0,C 180,E1 -6071.779,E2 -6071.779} C_VEL
LIN {X 0,Y 495.752,Z 381.358,A -85,B 0,C 180,E1 -6075.139,E2 -6075.139} C_VEL
LIN {X 0,Y 495.76,Z 381.358,A -85,B 0,C 180,E1 -6078.219,E2 -6078.219} C_VEL
LIN {X 0,Y 495.753,Z 381.358,A -85,B 0,C 180,E1 -6081.408,E2 -6081.408} C_VEL
LIN {X 0,Y 495.761,Z 381.359,A -85,B 0,C 180,E1 -6084.463,E2 -6084.463} C_VEL
LIN {X 0,Y 495.77,Z 381.357,A -85,B 0,C 180,E1 -6087.406,E2 -6087.406} C_VEL
LIN {X 0,Y 495.769,Z 381.353,A -85,B 0,C 180,E1 -6090.254,E2 -6090.254} C_VEL
LIN {X 0,Y 495.827,Z 381.346,A -85,B 0,C 180,E1 -6093.251,E2 -6093.251} C_VEL
LIN {X 0,Y 495.752,Z 381.359,A -85,B 0,C 180,E1 -6095.725,E2 -6095.725} C_VEL
LIN {X 0,Y 495.746,Z 381.357,A -85,B 0,C 180,E1 -6098.371,E2 -6098.371} C_VEL
LIN {X 0,Y 495.787,Z 381.353,A -85,B 0,C 180,E1 -6100.972,E2 -6100.972} C_VEL
LIN {X 0,Y 495.781,Z 381.354,A -85,B 0,C 180,E1 -6103.53,E2 -6103.53} C_VEL
LIN {X 0,Y 495.802,Z 381.349,A -85,B 0,C 180,E1 -6106.056,E2 -6106.056} C_VEL
LIN {X 0,Y 495.855,Z 381.347,A -85,B 0,C 180,E1 -6108.555,E2 -6108.555} C_VEL
LIN {X 0,Y 495.876,Z 381.344,A -85,B 0,C 180,E1 -6111.852,E2 -6111.852} C_VEL
LIN {X 0,Y 495.899,Z 381.337,A -85,B 0,C 180,E1 -6114.306,E2 -6114.306} C_VEL
LIN {X 0,Y 495.996,Z 381.325,A -85,B 0,C 180,E1 -6117.564,E2 -6117.564} C_VEL
LIN {X 0,Y 496.008,Z 381.323,A -85,B 0,C 180,E1 -6120.812,E2 -6120.812} C_VEL
LIN {X 0,Y 495.846,Z 381.348,A -85,B 0,C 180,E1 -6123.25,E2 -6123.25} C_VEL
LIN {X 0,Y 495.883,Z 381.344,A -85,B 0,C 180,E1 -6126.51,E2 -6126.51} C_VEL
LIN {X 0,Y 495.843,Z 381.344,A -85,B 0,C 180,E1 -6128.97,E2 -6128.97} C_VEL
LIN {X 0,Y 495.832,Z 381.345,A -85,B 0,C 180,E1 -6132.035,E2 -6132.035} C_VEL
LIN {X 0,Y 495.827,Z 381.346,A -85,B 0,C 180,E1 -6135.452,E2 -6135.452} C_VEL
LIN {X 0,Y 495.81,Z 381.35,A -85,B 0,C 180,E1 -6138.247,E2 -6138.247} C_VEL
LIN {X 0,Y 495.777,Z 381.354,A -85,B 0,C 180,E1 -6140.756,E2 -6140.756} C_VEL
LIN {X 0,Y 495.756,Z 381.353,A -85,B 0,C 180,E1 -6143.387,E2 -6143.387} C_VEL
LIN {X 0,Y 495.794,Z 381.354,A -85,B 0,C 180,E1 -6146.068,E2 -6146.068} C_VEL
LIN {X 0,Y 495.775,Z 381.354,A -85,B 0,C 180,E1 -6148.815,E2 -6148.815} C_VEL
LIN {X 0,Y 495.757,Z 381.355,A -85,B 0,C 180,E1 -6151.725,E2 -6151.725} C_VEL
LIN {X 0,Y 495.779,Z 381.353,A -85,B 0,C 180,E1 -6154.695,E2 -6154.695} C_VEL
LIN {X 0,Y 495.736,Z 381.362,A -85,B 0,C 180,E1 -6157.561,E2 -6157.561} C_VEL
LIN {X 0,Y 495.796,Z 381.353,A -85,B 0,C 180,E1 -6160.052,E2 -6160.052} C_VEL
LIN {X 0,Y 495.727,Z 381.36,A -85,B 0,C 180,E1 -6162.883,E2 -6162.883} C_VEL
LIN {X 0,Y 495.73,Z 381.361,A -85,B 0,C 180,E1 -6165.998,E2 -6165.998} C_VEL
LIN {X 0,Y 495.794,Z 381.456,A -85,B 0,C 180,E1 -6169.303,E2 -6169.303} C_VEL
LIN {X 0,Y 496.202,Z 385.154,A -85,B 0,C 180,E1 -6171.45,E2 -6171.45} C_VEL
LIN {X 0,Y 496.162,Z 389.487,A -85,B 0,C 180,E1 -6173.842,E2 -6173.842} C_VEL
LIN {X 0,Y 495.963,Z 394.94,A -85,B 0,C 180,E1 -6176.726,E2 -6176.726} C_VEL
LIN {X 0,Y 495.779,Z 401.029,A -85,B 0,C 180,E1 -6179.85,E2 -6179.85} C_VEL
LIN {X 0,Y 495.602,Z 407.99,A -85,B 0,C 180,E1 -6183.302,E2 -6183.302} C_VEL
LIN {X 0,Y 495.477,Z 412.975,A -85,B 0,C 180,E1 -6185.711,E2 -6185.711} C_VEL
LIN {X 0,Y 495.392,Z 418.563,A -85,B 0,C 180,E1 -6188.355,E2 -6188.355} C_VEL
LIN {X 0,Y 495.265,Z 424.158,A -85,B 0,C 180,E1 -6190.951,E2 -6190.951} C_VEL
LIN {X 0,Y 495.253,Z 427.47,A -85,B 0,C 180,E1 -6192.47,E2 -6192.47} C_VEL
LIN {X 0,Y 498.373,Z 442.288,A -85,B 0,C 180,E1 -6192.915,E2 -6192.915} C_VEL
LIN {X 0,Y 499.039,Z 446.232,A -85,B 0,C 180,E1 -6193.053,E2 -6193.053} C_VEL
LIN {X 0,Y 498.671,Z 459.048,A -85,B 0,C 180,E1 -6193.522,E2 -6193.522} C_VEL
LIN {X 0,Y 498.209,Z 471.749,A -85,B 0,C 180,E1 -6194.138,E2 -6194.138} C_VEL
LIN {X 0,Y 497.709,Z 484.91,A -85,B 0,C 180,E1 -6194.961,E2 -6194.961} C_VEL
LIN {X 0,Y 497.181,Z 496.811,A -85,B 0,C 180,E1 -6195.887,E2 -6195.887} C_VEL
LIN {X 0,Y 496.642,Z 507.681,A -85,B 0,C 180,E1 -6196.914,E2 -6196.914} C_VEL
LIN {X 0,Y 496.215,Z 518.63,A -85,B 0,C 180,E1 -6198.176,E2 -6198.176} C_VEL
LIN {X 0,Y 495.833,Z 527.287,A -85,B 0,C 180,E1 -6199.382,E2 -6199.382} C_VEL
LIN {X 0,Y 495.491,Z 535.782,A -85,B 0,C 180,E1 -6200.818,E2 -6200.818} C_VEL
LIN {X 0,Y 495.243,Z 542.627,A -85,B 0,C 180,E1 -6202.252,E2 -6202.252} C_VEL
LIN {X 0,Y 495.132,Z 548.296,A -85,B 0,C 180,E1 -6203.752,E2 -6203.752} C_VEL
LIN {X 0,Y 495.031,Z 552.232,A -85,B 0,C 180,E1 -6205.113,E2 -6205.113} C_VEL
LIN {X 0,Y 495.033,Z 555.63,A -85,B 0,C 180,E1 -6206.744,E2 -6206.744} C_VEL
LIN {X 0,Y 494.958,Z 557.64,A -85,B 0,C 180,E1 -6208.373,E2 -6208.373} C_VEL
LIN {X 0,Y 494.896,Z 558.306,A -85,B 0,C 180,E1 -6210,E2 -6210} C_VEL
LIN {X 0,Y 494.958,Z 557.641,A -85,B 0,C 180,E1 -6211.627,E2 -6211.627} C_VEL
LIN {X 0,Y 495.033,Z 555.635,A -85,B 0,C 180,E1 -6213.255,E2 -6213.255} C_VEL
LIN {X 0,Y 495.031,Z 552.236,A -85,B 0,C 180,E1 -6214.886,E2 -6214.886} C_VEL
LIN {X 0,Y 495.129,Z 548.305,A -85,B 0,C 180,E1 -6216.245,E2 -6216.245} C_VEL
LIN {X 0,Y 495.243,Z 542.627,A -85,B 0,C 180,E1 -6217.748,E2 -6217.748} C_VEL
LIN {X 0,Y 495.491,Z 535.784,A -85,B 0,C 180,E1 -6219.182,E2 -6219.182} C_VEL
LIN {X 0,Y 495.832,Z 527.288,A -85,B 0,C 180,E1 -6220.618,E2 -6220.618} C_VEL
LIN {X 0,Y 496.204,Z 517.543,A -85,B 0,C 180,E1 -6221.963,E2 -6221.963} C_VEL
LIN {X 0,Y 496.642,Z 507.682,A -85,B 0,C 180,E1 -6223.086,E2 -6223.086} C_VEL
LIN {X 0,Y 497.181,Z 496.813,A -85,B 0,C 180,E1 -6224.113,E2 -6224.113} C_VEL
LIN {X 0,Y 497.699,Z 484.916,A -85,B 0,C 180,E1 -6225.039,E2 -6225.039} C_VEL
LIN {X 0,Y 498.202,Z 471.748,A -85,B 0,C 180,E1 -6225.862,E2 -6225.862} C_VEL
LIN {X 0,Y 498.661,Z 457.734,A -85,B 0,C 180,E1 -6226.532,E2 -6226.532} C_VEL
LIN {X 0,Y 498.945,Z 445.255,A -85,B 0,C 180,E1 -6226.979,E2 -6226.979} C_VEL
LIN {X 0,Y 496.059,Z 431.323,A -85,B 0,C 180,E1 -6227.431,E2 -6227.431} C_VEL
LIN {X 0,Y 495.253,Z 427.442,A -85,B 0,C 180,E1 -6227.529,E2 -6227.529} C_VEL
LIN {X 0,Y 495.348,Z 420.427,A -85,B 0,C 180,E1 -6230.775,E2 -6230.775} C_VEL
LIN {X 0,Y 495.43,Z 414.836,A -85,B 0,C 180,E1 -6233.403,E2 -6233.403} C_VEL
LIN {X 0,Y 495.527,Z 409.254,A -85,B 0,C 180,E1 -6236.083,E2 -6236.083} C_VEL
LIN {X 0,Y 495.673,Z 403.678,A -85,B 0,C 180,E1 -6238.821,E2 -6238.821} C_VEL
LIN {X 0,Y 495.864,Z 397.889,A -85,B 0,C 180,E1 -6241.745,E2 -6241.745} C_VEL
LIN {X 0,Y 496.054,Z 392.143,A -85,B 0,C 180,E1 -6244.741,E2 -6244.741} C_VEL
LIN {X 0,Y 496.233,Z 386.984,A -85,B 0,C 180,E1 -6247.523,E2 -6247.523} C_VEL
LIN {X 0,Y 496.08,Z 383.294,A -85,B 0,C 180,E1 -6249.607,E2 -6249.607} C_VEL
LIN {X 0,Y 495.793,Z 381.359,A -85,B 0,C 180,E1 -6250.814,E2 -6250.814} C_VEL
LIN {X 0,Y 495.729,Z 381.361,A -85,B 0,C 180,E1 -6254.002,E2 -6254.002} C_VEL
LIN {X 0,Y 495.726,Z 381.361,A -85,B 0,C 180,E1 -6257.117,E2 -6257.117} C_VEL
LIN {X 0,Y 495.795,Z 381.352,A -85,B 0,C 180,E1 -6259.948,E2 -6259.948} C_VEL
LIN {X 0,Y 495.736,Z 381.362,A -85,B 0,C 180,E1 -6262.552,E2 -6262.552} C_VEL
LIN {X 0,Y 495.787,Z 381.353,A -85,B 0,C 180,E1 -6265.457,E2 -6265.457} C_VEL
LIN {X 0,Y 495.758,Z 381.355,A -85,B 0,C 180,E1 -6268.364,E2 -6268.364} C_VEL
LIN {X 0,Y 495.789,Z 381.351,A -85,B 0,C 180,E1 -6271.507,E2 -6271.507} C_VEL
LIN {X 0,Y 495.782,Z 381.356,A -85,B 0,C 180,E1 -6273.932,E2 -6273.932} C_VEL
LIN {X 0,Y 495.75,Z 381.359,A -85,B 0,C 180,E1 -6277.495,E2 -6277.495} C_VEL
LIN {X 0,Y 495.78,Z 381.353,A -85,B 0,C 180,E1 -6280.11,E2 -6280.11} C_VEL
LIN {X 0,Y 495.789,Z 381.351,A -85,B 0,C 180,E1 -6282.682,E2 -6282.682} C_VEL
LIN {X 0,Y 495.797,Z 381.353,A -85,B 0,C 180,E1 -6285.217,E2 -6285.217} C_VEL
LIN {X 0,Y 495.854,Z 381.347,A -85,B 0,C 180,E1 -6288.555,E2 -6288.555} C_VEL
LIN {X 0,Y 495.875,Z 381.345,A -85,B 0,C 180,E1 -6291.852,E2 -6291.852} C_VEL
LIN {X 0,Y 495.898,Z 381.337,A -85,B 0,C 180,E1 -6294.307,E2 -6294.307} C_VEL
LIN {X 0,Y 495.996,Z 381.325,A -85,B 0,C 180,E1 -6297.564,E2 -6297.564} C_VEL
LIN {X 0,Y 496.001,Z 381.329,A -85,B 0,C 180,E1 -6300,E2 -6300} C_VEL
LIN {X 0,Y 495.994,Z 381.325,A -85,B 0,C 180,E1 -6302.436,E2 -6302.436} C_VEL
LIN {X 0,Y 495.898,Z 381.337,A -85,B 0,C 180,E1 -6305.694,E2 -6305.694} C_VEL
LIN {X 0,Y 495.875,Z 381.345,A -85,B 0,C 180,E1 -6308.148,E2 -6308.148} C_VEL
LIN {X 0,Y 495.854,Z 381.348,A -85,B 0,C 180,E1 -6311.445,E2 -6311.445} C_VEL
LIN {X 0,Y 495.797,Z 381.354,A -85,B 0,C 180,E1 -6314.783,E2 -6314.783} C_VEL
LIN {X 0,Y 495.8,Z 381.352,A -85,B 0,C 180,E1 -6318.171,E2 -6318.171} C_VEL
LIN {X 0,Y 495.776,Z 381.354,A -85,B 0,C 180,E1 -6320.756,E2 -6320.756} C_VEL
LIN {X 0,Y 495.755,Z 381.355,A -85,B 0,C 180,E1 -6323.387,E2 -6323.387} C_VEL
LIN {X 0,Y 495.793,Z 381.355,A -85,B 0,C 180,E1 -6326.068,E2 -6326.068} C_VEL
LIN {X 0,Y 495.774,Z 381.354,A -85,B 0,C 180,E1 -6328.815,E2 -6328.815} C_VEL
LIN {X 0,Y 495.757,Z 381.355,A -85,B 0,C 180,E1 -6331.725,E2 -6331.725} C_VEL
LIN {X 0,Y 495.779,Z 381.352,A -85,B 0,C 180,E1 -6334.695,E2 -6334.695} C_VEL
LIN {X 0,Y 495.736,Z 381.36,A -85,B 0,C 180,E1 -6337.561,E2 -6337.561} C_VEL
LIN {X 0,Y 495.769,Z 381.358,A -85,B 0,C 180,E1 -6340.7,E2 -6340.7} C_VEL
LIN {X 0,Y 495.736,Z 381.361,A -85,B 0,C 180,E1 -6344.001,E2 -6344.001} C_VEL
LIN {X 0,Y 495.76,Z 381.359,A -85,B 0,C 180,E1 -6347.121,E2 -6347.121} C_VEL
LIN {X 0,Y 495.756,Z 381.36,A -85,B 0,C 180,E1 -6349.954,E2 -6349.954} C_VEL
LIN {X 0,Y 495.731,Z 381.408,A -85,B 0,C 180,E1 -6350.36,E2 -6350.36} C_VEL
LIN {X 0,Y 495.917,Z 384.682,A -85,B 0,C 180,E1 -6352.525,E2 -6352.525} C_VEL
LIN {X 0,Y 495.859,Z 389.309,A -85,B 0,C 180,E1 -6355.463,E2 -6355.463} C_VEL
LIN {X 0,Y 495.726,Z 394.035,A -85,B 0,C 180,E1 -6358.362,E2 -6358.362} C_VEL
LIN {X 0,Y 495.581,Z 397.691,A -85,B 0,C 180,E1 -6360.537,E2 -6360.537} C_VEL
LIN {X 0,Y 494.859,Z 398.899,A -85,B 0,C 180,E1 -6361.2,E2 -6361.2} C_VEL
LIN {X 0,Y 491.941,Z 401.052,A -85,B 0,C 180,E1 -6362.272,E2 -6362.272} C_VEL
LIN {X 0,Y 489.498,Z 402.79,A -85,B 0,C 180,E1 -6363.135,E2 -6363.135} C_VEL
LIN {X 0,Y 488.45,Z 404.048,A -85,B 0,C 180,E1 -6363.804,E2 -6363.804} C_VEL
LIN {X 0,Y 488.363,Z 404.447,A -85,B 0,C 180,E1 -6364.032,E2 -6364.032} C_VEL
LIN {X 0,Y 488.303,Z 408.263,A -85,B 0,C 180,E1 -6366.234,E2 -6366.234} C_VEL
LIN {X 0,Y 488.185,Z 413.773,A -85,B 0,C 180,E1 -6369.35,E2 -6369.35} C_VEL
LIN {X 0,Y 488.123,Z 418.989,A -85,B 0,C 180,E1 -6372.252,E2 -6372.252} C_VEL
LIN {X 0,Y 491.724,Z 434.938,A -85,B 0,C 180,E1 -6372.775,E2 -6372.775} C_VEL
LIN {X 0,Y 492.206,Z 438.109,A -85,B 0,C 180,E1 -6372.893,E2 -6372.893} C_VEL
LIN {X 0,Y 491.823,Z 451.174,A -85,B 0,C 180,E1 -6373.394,E2 -6373.394} C_VEL
LIN {X 0,Y 491.399,Z 463.547,A -85,B 0,C 180,E1 -6374.019,E2 -6374.019} C_VEL
LIN {X 0,Y 490.854,Z 476.48,A -85,B 0,C 180,E1 -6374.853,E2 -6374.853} C_VEL
LIN {X 0,Y 490.28,Z 488.201,A -85,B 0,C 180,E1 -6375.79,E2 -6375.79} C_VEL
LIN {X 0,Y 489.714,Z 499.021,A -85,B 0,C 180,E1 -6376.841,E2 -6376.841} C_VEL
LIN {X 0,Y 489.284,Z 509.28,A -85,B 0,C 180,E1 -6378.051,E2 -6378.051} C_VEL
LIN {X 0,Y 488.864,Z 517.611,A -85,B 0,C 180,E1 -6379.229,E2 -6379.229} C_VEL
LIN {X 0,Y 488.497,Z 526.123,A -85,B 0,C 180,E1 -6380.686,E2 -6380.686} C_VEL
LIN {X 0,Y 488.205,Z 532.98,A -85,B 0,C 180,E1 -6382.14,E2 -6382.14} C_VEL
LIN {X 0,Y 488.057,Z 539.009,A -85,B 0,C 180,E1 -6383.765,E2 -6383.765} C_VEL
LIN {X 0,Y 487.964,Z 542.62,A -85,B 0,C 180,E1 -6385.043,E2 -6385.043} C_VEL
LIN {X 0,Y 487.959,Z 546.036,A -85,B 0,C 180,E1 -6386.697,E2 -6386.697} C_VEL
LIN {X 0,Y 487.89,Z 548.068,A -85,B 0,C 180,E1 -6388.349,E2 -6388.349} C_VEL
LIN {X 0,Y 487.818,Z 548.77,A -85,B 0,C 180,E1 -6390,E2 -6390} C_VEL
LIN {X 0,Y 487.888,Z 548.148,A -85,B 0,C 180,E1 -6391.651,E2 -6391.651} C_VEL
LIN {X 0,Y 487.958,Z 546.189,A -85,B 0,C 180,E1 -6393.303,E2 -6393.303} C_VEL
LIN {X 0,Y 487.963,Z 542.847,A -85,B 0,C 180,E1 -6394.958,E2 -6394.958} C_VEL
LIN {X 0,Y 488.097,Z 538.024,A -85,B 0,C 180,E1 -6396.615,E2 -6396.615} C_VEL
LIN {X 0,Y 488.274,Z 531.566,A -85,B 0,C 180,E1 -6398.276,E2 -6398.276} C_VEL
LIN {X 0,Y 488.595,Z 524.374,A -85,B 0,C 180,E1 -6399.731,E2 -6399.731} C_VEL
LIN {X 0,Y 488.929,Z 516.839,A -85,B 0,C 180,E1 -6400.98,E2 -6400.98} C_VEL
LIN {X 0,Y 489.305,Z 507.757,A -85,B 0,C 180,E1 -6402.236,E2 -6402.236} C_VEL
LIN {X 0,Y 489.856,Z 496.83,A -85,B 0,C 180,E1 -6403.482,E2 -6403.482} C_VEL
LIN {X 0,Y 490.378,Z 485.657,A -85,B 0,C 180,E1 -6404.525,E2 -6404.525} C_VEL
LIN {X 0,Y 490.991,Z 473.294,A -85,B 0,C 180,E1 -6405.462,E2 -6405.462} C_VEL
LIN {X 0,Y 491.482,Z 461.396,A -85,B 0,C 180,E1 -6406.191,E2 -6406.191} C_VEL
LIN {X 0,Y 491.921,Z 448.317,A -85,B 0,C 180,E1 -6406.819,E2 -6406.819} C_VEL
LIN {X 0,Y 492.062,Z 436.604,A -85,B 0,C 180,E1 -6407.254,E2 -6407.254} C_VEL
LIN {X 0,Y 488.913,Z 422.543,A -85,B 0,C 180,E1 -6407.733,E2 -6407.733} C_VEL
LIN {X 0,Y 488.108,Z 418.983,A -85,B 0,C 180,E1 -6407.842,E2 -6407.842} C_VEL
LIN {X 0,Y 488.202,Z 413.14,A -85,B 0,C 180,E1 -6411.094,E2 -6411.094} C_VEL
LIN {X 0,Y 488.3,Z 408.421,A -85,B 0,C 180,E1 -6413.766,E2 -6413.766} C_VEL
LIN {X 0,Y 488.412,Z 403.081,A -85,B 0,C 180,E1 -6416.855,E2 -6416.855} C_VEL
LIN {X 0,Y 488.593,Z 397.391,A -85,B 0,C 180,E1 -6420.228,E2 -6420.228} C_VEL
LIN {X 0,Y 488.738,Z 392.643,A -85,B 0,C 180,E1 -6423.123,E2 -6423.123} C_VEL
LIN {X 0,Y 488.868,Z 387.498,A -85,B 0,C 180,E1 -6426.384,E2 -6426.384} C_VEL
LIN {X 0,Y 488.821,Z 383.423,A -85,B 0,C 180,E1 -6429.069,E2 -6429.069} C_VEL
LIN {X 0,Y 488.721,Z 382.238,A -85,B 0,C 180,E1 -6430.345,E2 -6430.345} C_VEL
LIN {X 0,Y 488.718,Z 382.236,A -85,B 0,C 180,E1 -6432.827,E2 -6432.827} C_VEL
LIN {X 0,Y 488.703,Z 382.237,A -85,B 0,C 180,E1 -6435.976,E2 -6435.976} C_VEL
LIN {X 0,Y 488.711,Z 382.234,A -85,B 0,C 180,E1 -6438.585,E2 -6438.585} C_VEL
LIN {X 0,Y 488.707,Z 382.237,A -85,B 0,C 180,E1 -6440.947,E2 -6440.947} C_VEL
LIN {X 0,Y 488.689,Z 382.236,A -85,B 0,C 180,E1 -6443.869,E2 -6443.869} C_VEL
LIN {X 0,Y 488.742,Z 382.229,A -85,B 0,C 180,E1 -6446.877,E2 -6446.877} C_VEL
LIN {X 0,Y 488.727,Z 382.231,A -85,B 0,C 180,E1 -6449.781,E2 -6449.781} C_VEL
LIN {X 0,Y 488.795,Z 382.223,A -85,B 0,C 180,E1 -6453.056,E2 -6453.056} C_VEL
LIN {X 0,Y 488.693,Z 382.234,A -85,B 0,C 180,E1 -6456.254,E2 -6456.254} C_VEL
LIN {X 0,Y 488.749,Z 382.229,A -85,B 0,C 180,E1 -6459.176,E2 -6459.176} C_VEL
LIN {X 0,Y 488.763,Z 382.227,A -85,B 0,C 180,E1 -6461.628,E2 -6461.628} C_VEL
LIN {X 0,Y 488.768,Z 382.226,A -85,B 0,C 180,E1 -6465,E2 -6465} C_VEL
LIN {X 0,Y 488.809,Z 382.223,A -85,B 0,C 180,E1 -6468.388,E2 -6468.388} C_VEL
LIN {X 0,Y 488.821,Z 382.221,A -85,B 0,C 180,E1 -6471.734,E2 -6471.734} C_VEL
LIN {X 0,Y 488.858,Z 382.214,A -85,B 0,C 180,E1 -6474.224,E2 -6474.224} C_VEL
LIN {X 0,Y 488.964,Z 382.201,A -85,B 0,C 180,E1 -6477.529,E2 -6477.529} C_VEL
LIN {X 0,Y 488.958,Z 382.201,A -85,B 0,C 180,E1 -6480.824,E2 -6480.824} C_VEL
LIN {X 0,Y 488.964,Z 382.201,A -85,B 0,C 180,E1 -6482.471,E2 -6482.471} C_VEL
LIN {X 0,Y 488.858,Z 382.213,A -85,B 0,C 180,E1 -6485.776,E2 -6485.776} C_VEL
LIN {X 0,Y 488.819,Z 382.223,A -85,B 0,C 180,E1 -6488.266,E2 -6488.266} C_VEL
LIN {X 0,Y 488.809,Z 382.223,A -85,B 0,C 180,E1 -6491.612,E2 -6491.612} C_VEL
LIN {X 0,Y 488.768,Z 382.227,A -85,B 0,C 180,E1 -6495,E2 -6495} C_VEL
LIN {X 0,Y 488.758,Z 382.227,A -85,B 0,C 180,E1 -6498.442,E2 -6498.442} C_VEL
LIN {X 0,Y 488.711,Z 382.237,A -85,B 0,C 180,E1 -6501.071,E2 -6501.071} C_VEL
LIN {X 0,Y 488.697,Z 382.233,A -85,B 0,C 180,E1 -6503.745,E2 -6503.745} C_VEL
LIN {X 0,Y 488.795,Z 382.221,A -85,B 0,C 180,E1 -6506.944,E2 -6506.944} C_VEL
LIN {X 0,Y 488.712,Z 382.232,A -85,B 0,C 180,E1 -6510.363,E2 -6510.363} C_VEL
LIN {X 0,Y 488.738,Z 382.23,A -85,B 0,C 180,E1 -6513.484,E2 -6513.484} C_VEL
LIN {X 0,Y 488.692,Z 382.237,A -85,B 0,C 180,E1 -6516.356,E2 -6516.356} C_VEL
LIN {X 0,Y 488.751,Z 382.232,A -85,B 0,C 180,E1 -6519.249,E2 -6519.249} C_VEL
LIN {X 0,Y 488.693,Z 382.238,A -85,B 0,C 180,E1 -6522.525,E2 -6522.525} C_VEL
LIN {X 0,Y 488.703,Z 382.238,A -85,B 0,C 180,E1 -6525.197,E2 -6525.197} C_VEL
LIN {X 0,Y 488.713,Z 382.237,A -85,B 0,C 180,E1 -6528.4,E2 -6528.4} C_VEL
LIN {X 0,Y 488.782,Z 382.356,A -85,B 0,C 180,E1 -6529.139,E2 -6529.139} C_VEL
LIN {X 0,Y 489.137,Z 385.288,A -85,B 0,C 180,E1 -6530.885,E2 -6530.885} C_VEL
LIN {X 0,Y 489.153,Z 390.063,A -85,B 0,C 180,E1 -6533.571,E2 -6533.571} C_VEL
LIN {X 0,Y 488.941,Z 395.457,A -85,B 0,C 180,E1 -6536.479,E2 -6536.479} C_VEL
LIN {X 0,Y 488.743,Z 401.783,A -85,B 0,C 180,E1 -6539.782,E2 -6539.782} C_VEL
LIN {X 0,Y 488.542,Z 408.401,A -85,B 0,C 180,E1 -6543.114,E2 -6543.114} C_VEL
LIN {X 0,Y 488.383,Z 414.786,A -85,B 0,C 180,E1 -6546.238,E2 -6546.238} C_VEL
LIN {X 0,Y 488.285,Z 421.229,A -85,B 0,C 180,E1 -6549.319,E2 -6549.319} C_VEL
LIN {X 0,Y 488.19,Z 427.572,A -85,B 0,C 180,E1 -6552.213,E2 -6552.213} C_VEL
LIN {X 0,Y 491.317,Z 442.049,A -85,B 0,C 180,E1 -6552.657,E2 -6552.657} C_VEL
LIN {X 0,Y 492.191,Z 447.179,A -85,B 0,C 180,E1 -6552.845,E2 -6552.845} C_VEL
LIN {X 0,Y 491.812,Z 460.26,A -85,B 0,C 180,E1 -6553.345,E2 -6553.345} C_VEL
LIN {X 0,Y 491.29,Z 473.455,A -85,B 0,C 180,E1 -6554.016,E2 -6554.016} C_VEL
LIN {X 0,Y 490.74,Z 486.268,A -85,B 0,C 180,E1 -6554.849,E2 -6554.849} C_VEL
LIN {X 0,Y 490.217,Z 497.918,A -85,B 0,C 180,E1 -6555.788,E2 -6555.788} C_VEL
LIN {X 0,Y 489.696,Z 507.611,A -85,B 0,C 180,E1 -6556.725,E2 -6556.725} C_VEL
LIN {X 0,Y 489.215,Z 517.861,A -85,B 0,C 180,E1 -6557.914,E2 -6557.914} C_VEL
LIN {X 0,Y 488.818,Z 527.218,A -85,B 0,C 180,E1 -6559.227,E2 -6559.227} C_VEL
LIN {X 0,Y 488.435,Z 535.713,A -85,B 0,C 180,E1 -6560.684,E2 -6560.684} C_VEL
LIN {X 0,Y 488.175,Z 542.558,A -85,B 0,C 180,E1 -6562.139,E2 -6562.139} C_VEL
LIN {X 0,Y 488.076,Z 547.65,A -85,B 0,C 180,E1 -6563.494,E2 -6563.494} C_VEL
LIN {X 0,Y 487.962,Z 552.163,A -85,B 0,C 180,E1 -6565.042,E2 -6565.042} C_VEL
LIN {X 0,Y 487.955,Z 555.562,A -85,B 0,C 180,E1 -6566.697,E2 -6566.697} C_VEL
LIN {X 0,Y 487.886,Z 557.571,A -85,B 0,C 180,E1 -6568.349,E2 -6568.349} C_VEL
LIN {X 0,Y 487.817,Z 558.237,A -85,B 0,C 180,E1 -6570,E2 -6570} C_VEL
LIN {X 0,Y 487.886,Z 557.573,A -85,B 0,C 180,E1 -6571.651,E2 -6571.651} C_VEL
LIN {X 0,Y 487.955,Z 555.566,A -85,B 0,C 180,E1 -6573.303,E2 -6573.303} C_VEL
LIN {X 0,Y 487.962,Z 552.167,A -85,B 0,C 180,E1 -6574.957,E2 -6574.957} C_VEL
LIN {X 0,Y 488.095,Z 547.275,A -85,B 0,C 180,E1 -6576.615,E2 -6576.615} C_VEL
LIN {X 0,Y 488.258,Z 540.745,A -85,B 0,C 180,E1 -6578.276,E2 -6578.276} C_VEL
LIN {X 0,Y 488.565,Z 533.479,A -85,B 0,C 180,E1 -6579.731,E2 -6579.731} C_VEL
LIN {X 0,Y 488.945,Z 524.479,A -85,B 0,C 180,E1 -6581.189,E2 -6581.189} C_VEL
LIN {X 0,Y 489.347,Z 515.032,A -85,B 0,C 180,E1 -6582.441,E2 -6582.441} C_VEL
LIN {X 0,Y 489.834,Z 504.574,A -85,B 0,C 180,E1 -6583.588,E2 -6583.588} C_VEL
LIN {X 0,Y 490.383,Z 493.033,A -85,B 0,C 180,E1 -6584.631,E2 -6584.631} C_VEL
LIN {X 0,Y 491.02,Z 480.23,A -85,B 0,C 180,E1 -6585.567,E2 -6585.567} C_VEL
LIN {X 0,Y 491.515,Z 467.724,A -85,B 0,C 180,E1 -6586.297,E2 -6586.297} C_VEL
LIN {X 0,Y 491.955,Z 453.819,A -85,B 0,C 180,E1 -6586.922,E2 -6586.922} C_VEL
LIN {X 0,Y 492.027,Z 445.913,A -85,B 0,C 180,E1 -6587.204,E2 -6587.204} C_VEL
LIN {X 0,Y 489.031,Z 431.362,A -85,B 0,C 180,E1 -6587.688,E2 -6587.688} C_VEL
LIN {X 0,Y 488.198,Z 427.374,A -85,B 0,C 180,E1 -6587.803,E2 -6587.803} C_VEL
LIN {X 0,Y 488.283,Z 420.363,A -85,B 0,C 180,E1 -6591.09,E2 -6591.09} C_VEL
LIN {X 0,Y 488.385,Z 414.784,A -85,B 0,C 180,E1 -6593.761,E2 -6593.761} C_VEL
LIN {X 0,Y 488.543,Z 408.398,A -85,B 0,C 180,E1 -6596.886,E2 -6596.886} C_VEL
LIN {X 0,Y 488.742,Z 401.778,A -85,B 0,C 180,E1 -6600.218,E2 -6600.218} C_VEL
LIN {X 0,Y 488.94,Z 395.451,A -85,B 0,C 180,E1 -6603.52,E2 -6603.52} C_VEL
LIN {X 0,Y 489.152,Z 390.054,A -85,B 0,C 180,E1 -6606.429,E2 -6606.429} C_VEL
LIN {X 0,Y 489.141,Z 385.283,A -85,B 0,C 180,E1 -6609.116,E2 -6609.116} C_VEL
LIN {X 0,Y 488.753,Z 382.235,A -85,B 0,C 180,E1 -6611,E2 -6611} C_VEL
LIN {X 0,Y 488.695,Z 382.237,A -85,B 0,C 180,E1 -6614.023,E2 -6614.023} C_VEL
LIN {X 0,Y 488.71,Z 382.235,A -85,B 0,C 180,E1 -6617.174,E2 -6617.174} C_VEL
LIN {X 0,Y 488.738,Z 382.233,A -85,B 0,C 180,E1 -6619.677,E2 -6619.677} C_VEL
LIN {X 0,Y 488.686,Z 382.238,A -85,B 0,C 180,E1 -6622.277,E2 -6622.277} C_VEL
LIN {X 0,Y 488.73,Z 382.231,A -85,B 0,C 180,E1 -6625.051,E2 -6625.051} C_VEL
LIN {X 0,Y 488.705,Z 382.235,A -85,B 0,C 180,E1 -6628.046,E2 -6628.046} C_VEL
LIN {X 0,Y 488.725,Z 382.236,A -85,B 0,C 180,E1 -6630.73,E2 -6630.73} C_VEL
LIN {X 0,Y 488.754,Z 382.228,A -85,B 0,C 180,E1 -6633.528,E2 -6633.528} C_VEL
LIN {X 0,Y 488.678,Z 382.237,A -85,B 0,C 180,E1 -6636.254,E2 -6636.254} C_VEL
LIN {X 0,Y 488.748,Z 382.231,A -85,B 0,C 180,E1 -6639.176,E2 -6639.176} C_VEL
LIN {X 0,Y 488.761,Z 382.227,A -85,B 0,C 180,E1 -6641.628,E2 -6641.628} C_VEL
LIN {X 0,Y 488.767,Z 382.227,A -85,B 0,C 180,E1 -6645,E2 -6645} C_VEL
LIN {X 0,Y 488.808,Z 382.223,A -85,B 0,C 180,E1 -6648.388,E2 -6648.388} C_VEL
LIN {X 0,Y 488.819,Z 382.223,A -85,B 0,C 180,E1 -6651.734,E2 -6651.734} C_VEL
LIN {X 0,Y 488.857,Z 382.214,A -85,B 0,C 180,E1 -6654.224,E2 -6654.224} C_VEL
LIN {X 0,Y 488.963,Z 382.201,A -85,B 0,C 180,E1 -6657.529,E2 -6657.529} C_VEL
LIN {X 0,Y 488.956,Z 382.202,A -85,B 0,C 180,E1 -6660.824,E2 -6660.824} C_VEL
LIN {X 0,Y 488.962,Z 382.201,A -85,B 0,C 180,E1 -6662.471,E2 -6662.471} C_VEL
LIN {X 0,Y 488.857,Z 382.214,A -85,B 0,C 180,E1 -6665.776,E2 -6665.776} C_VEL
LIN {X 0,Y 488.819,Z 382.223,A -85,B 0,C 180,E1 -6668.266,E2 -6668.266} C_VEL
LIN {X 0,Y 488.808,Z 382.223,A -85,B 0,C 180,E1 -6671.612,E2 -6671.612} C_VEL
LIN {X 0,Y 488.767,Z 382.227,A -85,B 0,C 180,E1 -6675,E2 -6675} C_VEL
LIN {X 0,Y 488.757,Z 382.227,A -85,B 0,C 180,E1 -6678.442,E2 -6678.442} C_VEL
LIN {X 0,Y 488.71,Z 382.238,A -85,B 0,C 180,E1 -6681.071,E2 -6681.071} C_VEL
LIN {X 0,Y 488.696,Z 382.235,A -85,B 0,C 180,E1 -6683.745,E2 -6683.745} C_VEL
LIN {X 0,Y 488.794,Z 382.222,A -85,B 0,C 180,E1 -6686.944,E2 -6686.944} C_VEL
LIN {X 0,Y 488.711,Z 382.233,A -85,B 0,C 180,E1 -6690.363,E2 -6690.363} C_VEL
LIN {X 0,Y 488.738,Z 382.23,A -85,B 0,C 180,E1 -6693.485,E2 -6693.485} C_VEL
LIN {X 0,Y 488.692,Z 382.235,A -85,B 0,C 180,E1 -6696.356,E2 -6696.356} C_VEL
LIN {X 0,Y 488.704,Z 382.236,A -85,B 0,C 180,E1 -6699.254,E2 -6699.254} C_VEL
LIN {X 0,Y 488.71,Z 382.233,A -85,B 0,C 180,E1 -6701.6,E2 -6701.6} C_VEL
LIN {X 0,Y 488.714,Z 382.233,A -85,B 0,C 180,E1 -6704.801,E2 -6704.801} C_VEL
LIN {X 0,Y 488.698,Z 382.237,A -85,B 0,C 180,E1 -6707.475,E2 -6707.475} C_VEL
LIN {X 0,Y 488.735,Z 382.233,A -85,B 0,C 180,E1 -6709.677,E2 -6709.677} C_VEL
LIN {X 0,Y 488.782,Z 383.292,A -85,B 0,C 180,E1 -6710.936,E2 -6710.936} C_VEL
LIN {X 0,Y 488.869,Z 387.35,A -85,B 0,C 180,E1 -6713.616,E2 -6713.616} C_VEL
LIN {X 0,Y 488.742,Z 392.492,A -85,B 0,C 180,E1 -6716.877,E2 -6716.877} C_VEL
LIN {X 0,Y 488.592,Z 397.238,A -85,B 0,C 180,E1 -6719.772,E2 -6719.772} C_VEL
LIN {X 0,Y 488.418,Z 401.968,A -85,B 0,C 180,E1 -6722.583,E2 -6722.583} C_VEL
LIN {X 0,Y 488.363,Z 404.447,A -85,B 0,C 180,E1 -6724.032,E2 -6724.032} C_VEL
LIN {X 0,Y 487.679,Z 405.678,A -85,B 0,C 180,E1 -6724.704,E2 -6724.704} C_VEL
LIN {X 0,Y 484.768,Z 407.849,A -85,B 0,C 180,E1 -6725.791,E2 -6725.791} C_VEL
LIN {X 0,Y 482.312,Z 409.602,A -85,B 0,C 180,E1 -6726.666,E2 -6726.666} C_VEL
LIN {X 0,Y 481.261,Z 410.88,A -85,B 0,C 180,E1 -6727.345,E2 -6727.345} C_VEL
LIN {X 0,Y 481.178,Z 411.285,A -85,B 0,C 180,E1 -6727.575,E2 -6727.575} C_VEL
LIN {X 0,Y 481.07,Z 416.186,A -85,B 0,C 180,E1 -6730.366,E2 -6730.366} C_VEL
LIN {X 0,Y 481.051,Z 419.076,A -85,B 0,C 180,E1 -6731.992,E2 -6731.992} C_VEL
LIN {X 0,Y 484.539,Z 434.045,A -85,B 0,C 180,E1 -6732.482,E2 -6732.482} C_VEL
LIN {X 0,Y 485.386,Z 439.15,A -85,B 0,C 180,E1 -6732.679,E2 -6732.679} C_VEL
LIN {X 0,Y 484.979,Z 452.386,A -85,B 0,C 180,E1 -6733.207,E2 -6733.207} C_VEL
LIN {X 0,Y 484.499,Z 465.392,A -85,B 0,C 180,E1 -6733.894,E2 -6733.894} C_VEL
LIN {X 0,Y 483.916,Z 477.981,A -85,B 0,C 180,E1 -6734.738,E2 -6734.738} C_VEL
LIN {X 0,Y 483.311,Z 489.449,A -85,B 0,C 180,E1 -6735.688,E2 -6735.688} C_VEL
LIN {X 0,Y 482.715,Z 499.973,A -85,B 0,C 180,E1 -6736.744,E2 -6736.744} C_VEL
LIN {X 0,Y 482.295,Z 509.591,A -85,B 0,C 180,E1 -6737.906,E2 -6737.906} C_VEL
LIN {X 0,Y 481.779,Z 519.036,A -85,B 0,C 180,E1 -6739.281,E2 -6739.281} C_VEL
LIN {X 0,Y 481.404,Z 527.297,A -85,B 0,C 180,E1 -6740.759,E2 -6740.759} C_VEL
LIN {X 0,Y 481.15,Z 533.052,A -85,B 0,C 180,E1 -6742.024,E2 -6742.024} C_VEL
LIN {X 0,Y 481.034,Z 538.373,A -85,B 0,C 180,E1 -6743.462,E2 -6743.462} C_VEL
LIN {X 0,Y 480.9,Z 542.69,A -85,B 0,C 180,E1 -6744.97,E2 -6744.97} C_VEL
LIN {X 0,Y 480.884,Z 546.106,A -85,B 0,C 180,E1 -6746.649,E2 -6746.649} C_VEL
LIN {X 0,Y 480.791,Z 548.137,A -85,B 0,C 180,E1 -6748.325,E2 -6748.325} C_VEL
LIN {X 0,Y 480.742,Z 548.838,A -85,B 0,C 180,E1 -6750,E2 -6750} C_VEL
LIN {X 0,Y 480.79,Z 548.216,A -85,B 0,C 180,E1 -6751.675,E2 -6751.675} C_VEL
LIN {X 0,Y 480.883,Z 546.257,A -85,B 0,C 180,E1 -6753.351,E2 -6753.351} C_VEL
LIN {X 0,Y 480.897,Z 542.914,A -85,B 0,C 180,E1 -6755.031,E2 -6755.031} C_VEL
LIN {X 0,Y 481.012,Z 538.091,A -85,B 0,C 180,E1 -6756.713,E2 -6756.713} C_VEL
LIN {X 0,Y 481.232,Z 531.632,A -85,B 0,C 180,E1 -6758.398,E2 -6758.398} C_VEL
LIN {X 0,Y 481.559,Z 524.44,A -85,B 0,C 180,E1 -6759.874,E2 -6759.874} C_VEL
LIN {X 0,Y 481.942,Z 516.904,A -85,B 0,C 180,E1 -6761.141,E2 -6761.141} C_VEL
LIN {X 0,Y 482.302,Z 508.413,A -85,B 0,C 180,E1 -6762.338,E2 -6762.338} C_VEL
LIN {X 0,Y 482.799,Z 498.842,A -85,B 0,C 180,E1 -6763.468,E2 -6763.468} C_VEL
LIN {X 0,Y 483.377,Z 488.085,A -85,B 0,C 180,E1 -6764.525,E2 -6764.525} C_VEL
LIN {X 0,Y 483.982,Z 476.316,A -85,B 0,C 180,E1 -6765.476,E2 -6765.476} C_VEL
LIN {X 0,Y 484.584,Z 463.33,A -85,B 0,C 180,E1 -6766.32,E2 -6766.32} C_VEL
LIN {X 0,Y 485.071,Z 450.884,A -85,B 0,C 180,E1 -6766.953,E2 -6766.953} C_VEL
LIN {X 0,Y 485.28,Z 437.871,A -85,B 0,C 180,E1 -6767.461,E2 -6767.461} C_VEL
LIN {X 0,Y 482.243,Z 424.071,A -85,B 0,C 180,E1 -6767.957,E2 -6767.957} C_VEL
LIN {X 0,Y 481.053,Z 419.046,A -85,B 0,C 180,E1 -6768.115,E2 -6768.115} C_VEL
LIN {X 0,Y 481.123,Z 413.196,A -85,B 0,C 180,E1 -6771.419,E2 -6771.419} C_VEL
LIN {X 0,Y 481.256,Z 408.481,A -85,B 0,C 180,E1 -6774.136,E2 -6774.136} C_VEL
LIN {X 0,Y 481.363,Z 403.523,A -85,B 0,C 180,E1 -6777.049,E2 -6777.049} C_VEL
LIN {X 0,Y 481.497,Z 399.012,A -85,B 0,C 180,E1 -6779.754,E2 -6779.754} C_VEL
LIN {X 0,Y 481.667,Z 394.266,A -85,B 0,C 180,E1 -6782.675,E2 -6782.675} C_VEL
LIN {X 0,Y 481.776,Z 389.525,A -85,B 0,C 180,E1 -6785.698,E2 -6785.698} C_VEL
LIN {X 0,Y 481.838,Z 385.973,A -85,B 0,C 180,E1 -6788.035,E2 -6788.035} C_VEL
LIN {X 0,Y 481.672,Z 383.195,A -85,B 0,C 180,E1 -6789.941,E2 -6789.941} C_VEL
LIN {X 0,Y 481.669,Z 383.115,A -85,B 0,C 180,E1 -6793.297,E2 -6793.297} C_VEL
LIN {X 0,Y 481.661,Z 383.112,A -85,B 0,C 180,E1 -6795.641,E2 -6795.641} C_VEL
LIN {X 0,Y 481.659,Z 383.113,A -85,B 0,C 180,E1 -6798.958,E2 -6798.958} C_VEL
LIN {X 0,Y 481.659,Z 383.111,A -85,B 0,C 180,E1 -6801.993,E2 -6801.993} C_VEL
LIN {X 0,Y 481.696,Z 383.107,A -85,B 0,C 180,E1 -6805.318,E2 -6805.318} C_VEL
LIN {X 0,Y 481.648,Z 383.112,A -85,B 0,C 180,E1 -6808.312,E2 -6808.312} C_VEL
LIN {X 0,Y 481.703,Z 383.107,A -85,B 0,C 180,E1 -6811.219,E2 -6811.219} C_VEL
LIN {X 0,Y 481.704,Z 383.11,A -85,B 0,C 180,E1 -6814.043,E2 -6814.043} C_VEL
LIN {X 0,Y 481.677,Z 383.108,A -85,B 0,C 180,E1 -6816.812,E2 -6816.812} C_VEL
LIN {X 0,Y 481.699,Z 383.104,A -85,B 0,C 180,E1 -6819.503,E2 -6819.503} C_VEL
LIN {X 0,Y 481.708,Z 383.11,A -85,B 0,C 180,E1 -6822.158,E2 -6822.158} C_VEL
LIN {X 0,Y 481.748,Z 383.099,A -85,B 0,C 180,E1 -6824.776,E2 -6824.776} C_VEL
LIN {X 0,Y 481.754,Z 383.1,A -85,B 0,C 180,E1 -6828.215,E2 -6828.215} C_VEL
LIN {X 0,Y 481.766,Z 383.099,A -85,B 0,C 180,E1 -6831.612,E2 -6831.612} C_VEL
LIN {X 0,Y 481.819,Z 383.091,A -85,B 0,C 180,E1 -6834.14,E2 -6834.14} C_VEL
LIN {X 0,Y 481.93,Z 383.077,A -85,B 0,C 180,E1 -6837.492,E2 -6837.492} C_VEL
LIN {X 0,Y 481.909,Z 383.079,A -85,B 0,C 180,E1 -6840.836,E2 -6840.836} C_VEL
LIN {X 0,Y 481.931,Z 383.077,A -85,B 0,C 180,E1 -6842.507,E2 -6842.507} C_VEL
LIN {X 0,Y 481.819,Z 383.09,A -85,B 0,C 180,E1 -6845.86,E2 -6845.86} C_VEL
LIN {X 0,Y 481.765,Z 383.101,A -85,B 0,C 180,E1 -6848.388,E2 -6848.388} C_VEL
LIN {X 0,Y 481.754,Z 383.1,A -85,B 0,C 180,E1 -6851.785,E2 -6851.785} C_VEL
LIN {X 0,Y 481.747,Z 383.1,A -85,B 0,C 180,E1 -6855.224,E2 -6855.224} C_VEL
LIN {X 0,Y 481.716,Z 383.104,A -85,B 0,C 180,E1 -6858.722,E2 -6858.722} C_VEL
LIN {X 0,Y 481.651,Z 383.115,A -85,B 0,C 180,E1 -6861.394,E2 -6861.394} C_VEL
LIN {X 0,Y 481.68,Z 383.109,A -85,B 0,C 180,E1 -6864.113,E2 -6864.113} C_VEL
LIN {X 0,Y 481.75,Z 383.1,A -85,B 0,C 180,E1 -6867.139,E2 -6867.139} C_VEL
LIN {X 0,Y 481.681,Z 383.107,A -85,B 0,C 180,E1 -6869.741,E2 -6869.741} C_VEL
LIN {X 0,Y 481.674,Z 383.113,A -85,B 0,C 180,E1 -6872.674,E2 -6872.674} C_VEL
LIN {X 0,Y 481.646,Z 383.119,A -85,B 0,C 180,E1 -6875.709,E2 -6875.709} C_VEL
LIN {X 0,Y 481.722,Z 383.107,A -85,B 0,C 180,E1 -6879.355,E2 -6879.355} C_VEL
LIN {X 0,Y 481.651,Z 383.118,A -85,B 0,C 180,E1 -6882.16,E2 -6882.16} C_VEL
LIN {X 0,Y 481.656,Z 383.117,A -85,B 0,C 180,E1 -6885.542,E2 -6885.542} C_VEL
LIN {X 0,Y 481.73,Z 383.252,A -85,B 0,C 180,E1 -6888.966,E2 -6888.966} C_VEL
LIN {X 0,Y 482.134,Z 386.938,A -85,B 0,C 180,E1 -6891.185,E2 -6891.185} C_VEL
LIN {X 0,Y 482.156,Z 390.641,A -85,B 0,C 180,E1 -6893.3,E2 -6893.3} C_VEL
LIN {X 0,Y 481.923,Z 396.198,A -85,B 0,C 180,E1 -6896.347,E2 -6896.347} C_VEL
LIN {X 0,Y 481.706,Z 401.959,A -85,B 0,C 180,E1 -6899.406,E2 -6899.406} C_VEL
LIN {X 0,Y 481.52,Z 407.306,A -85,B 0,C 180,E1 -6902.157,E2 -6902.157} C_VEL
LIN {X 0,Y 481.376,Z 412.873,A -85,B 0,C 180,E1 -6904.951,E2 -6904.951} C_VEL
LIN {X 0,Y 481.24,Z 418.446,A -85,B 0,C 180,E1 -6907.685,E2 -6907.685} C_VEL
LIN {X 0,Y 481.134,Z 424.027,A -85,B 0,C 180,E1 -6910.369,E2 -6910.369} C_VEL
LIN {X 0,Y 481.126,Z 427.334,A -85,B 0,C 180,E1 -6911.939,E2 -6911.939} C_VEL
LIN {X 0,Y 484.169,Z 441.397,A -85,B 0,C 180,E1 -6912.375,E2 -6912.375} C_VEL
LIN {X 0,Y 485.351,Z 448.788,A -85,B 0,C 180,E1 -6912.656,E2 -6912.656} C_VEL
LIN {X 0,Y 484.904,Z 462.456,A -85,B 0,C 180,E1 -6913.21,E2 -6913.21} C_VEL
LIN {X 0,Y 484.383,Z 475.188,A -85,B 0,C 180,E1 -6913.892,E2 -6913.892} C_VEL
LIN {X 0,Y 483.783,Z 487.626,A -85,B 0,C 180,E1 -6914.734,E2 -6914.734} C_VEL
LIN {X 0,Y 483.238,Z 499.023,A -85,B 0,C 180,E1 -6915.686,E2 -6915.686} C_VEL
LIN {X 0,Y 482.647,Z 509.495,A -85,B 0,C 180,E1 -6916.742,E2 -6916.742} C_VEL
LIN {X 0,Y 482.186,Z 519.146,A -85,B 0,C 180,E1 -6917.912,E2 -6917.912} C_VEL
LIN {X 0,Y 481.724,Z 528.504,A -85,B 0,C 180,E1 -6919.28,E2 -6919.28} C_VEL
LIN {X 0,Y 481.34,Z 536.731,A -85,B 0,C 180,E1 -6920.758,E2 -6920.758} C_VEL
LIN {X 0,Y 481.126,Z 542.489,A -85,B 0,C 180,E1 -6922.023,E2 -6922.023} C_VEL
LIN {X 0,Y 480.972,Z 548.015,A -85,B 0,C 180,E1 -6923.525,E2 -6923.525} C_VEL
LIN {X 0,Y 480.897,Z 552.095,A -85,B 0,C 180,E1 -6924.969,E2 -6924.969} C_VEL
LIN {X 0,Y 480.861,Z 555.493,A -85,B 0,C 180,E1 -6926.648,E2 -6926.648} C_VEL
LIN {X 0,Y 480.787,Z 557.502,A -85,B 0,C 180,E1 -6928.325,E2 -6928.325} C_VEL
LIN {X 0,Y 480.741,Z 558.168,A -85,B 0,C 180,E1 -6930,E2 -6930} C_VEL
LIN {X 0,Y 480.787,Z 557.504,A -85,B 0,C 180,E1 -6931.675,E2 -6931.675} C_VEL
LIN {X 0,Y 480.861,Z 555.497,A -85,B 0,C 180,E1 -6933.351,E2 -6933.351} C_VEL
LIN {X 0,Y 480.896,Z 552.098,A -85,B 0,C 180,E1 -6935.03,E2 -6935.03} C_VEL
LIN {X 0,Y 481.007,Z 547.206,A -85,B 0,C 180,E1 -6936.712,E2 -6936.712} C_VEL
LIN {X 0,Y 481.212,Z 540.676,A -85,B 0,C 180,E1 -6938.398,E2 -6938.398} C_VEL
LIN {X 0,Y 481.494,Z 533.409,A -85,B 0,C 180,E1 -6939.875,E2 -6939.875} C_VEL
LIN {X 0,Y 481.948,Z 524.41,A -85,B 0,C 180,E1 -6941.354,E2 -6941.354} C_VEL
LIN {X 0,Y 482.366,Z 514.963,A -85,B 0,C 180,E1 -6942.624,E2 -6942.624} C_VEL
LIN {X 0,Y 482.892,Z 504.505,A -85,B 0,C 180,E1 -6943.787,E2 -6943.787} C_VEL
LIN {X 0,Y 483.495,Z 492.964,A -85,B 0,C 180,E1 -6944.844,E2 -6944.844} C_VEL
LIN {X 0,Y 484.163,Z 480.161,A -85,B 0,C 180,E1 -6945.793,E2 -6945.793} C_VEL
LIN {X 0,Y 484.681,Z 467.944,A -85,B 0,C 180,E1 -6946.517,E2 -6946.517} C_VEL
LIN {X 0,Y 485.147,Z 453.75,A -85,B 0,C 180,E1 -6947.167,E2 -6947.167} C_VEL
LIN {X 0,Y 485.274,Z 447.303,A -85,B 0,C 180,E1 -6947.4,E2 -6947.4} C_VEL
LIN {X 0,Y 482.339,Z 432.928,A -85,B 0,C 180,E1 -6947.909,E2 -6947.909} C_VEL
LIN {X 0,Y 481.126,Z 427.334,A -85,B 0,C 180,E1 -6948.06,E2 -6948.06} C_VEL
LIN {X 0,Y 481.222,Z 420.305,A -85,B 0,C 180,E1 -6951.414,E2 -6951.414} C_VEL
LIN {X 0,Y 481.354,Z 414.723,A -85,B 0,C 180,E1 -6954.13,E2 -6954.13} C_VEL
LIN {X 0,Y 481.502,Z 408.797,A -85,B 0,C 180,E1 -6957.082,E2 -6957.082} C_VEL
LIN {X 0,Y 481.706,Z 401.953,A -85,B 0,C 180,E1 -6960.593,E2 -6960.593} C_VEL
LIN {X 0,Y 481.929,Z 395.966,A -85,B 0,C 180,E1 -6963.774,E2 -6963.774} C_VEL
LIN {X 0,Y 482.147,Z 390.622,A -85,B 0,C 180,E1 -6966.707,E2 -6966.707} C_VEL
LIN {X 0,Y 482.136,Z 386.937,A -85,B 0,C 180,E1 -6968.815,E2 -6968.815} C_VEL
LIN {X 0,Y 481.719,Z 383.111,A -85,B 0,C 180,E1 -6971.174,E2 -6971.174} C_VEL
LIN {X 0,Y 481.655,Z 383.117,A -85,B 0,C 180,E1 -6974.458,E2 -6974.458} C_VEL
LIN {X 0,Y 481.65,Z 383.119,A -85,B 0,C 180,E1 -6977.84,E2 -6977.84} C_VEL
LIN {X 0,Y 481.721,Z 383.106,A -85,B 0,C 180,E1 -6980.645,E2 -6980.645} C_VEL
LIN {X 0,Y 481.645,Z 383.118,A -85,B 0,C 180,E1 -6984.291,E2 -6984.291} C_VEL
LIN {X 0,Y 481.674,Z 383.113,A -85,B 0,C 180,E1 -6987.326,E2 -6987.326} C_VEL
LIN {X 0,Y 481.68,Z 383.11,A -85,B 0,C 180,E1 -6990.259,E2 -6990.259} C_VEL
LIN {X 0,Y 481.747,Z 383.1,A -85,B 0,C 180,E1 -6993.112,E2 -6993.112} C_VEL
LIN {X 0,Y 481.66,Z 383.114,A -85,B 0,C 180,E1 -6995.886,E2 -6995.886} C_VEL
LIN {X 0,Y 481.704,Z 383.11,A -85,B 0,C 180,E1 -6999.028,E2 -6999.028} C_VEL
LIN {X 0,Y 481.709,Z 383.108,A -85,B 0,C 180,E1 -7002.159,E2 -7002.159} C_VEL
LIN {X 0,Y 481.746,Z 383.1,A -85,B 0,C 180,E1 -7004.776,E2 -7004.776} C_VEL
LIN {X 0,Y 481.753,Z 383.1,A -85,B 0,C 180,E1 -7008.215,E2 -7008.215} C_VEL
LIN {X 0,Y 481.765,Z 383.1,A -85,B 0,C 180,E1 -7011.612,E2 -7011.612} C_VEL
LIN {X 0,Y 481.818,Z 383.091,A -85,B 0,C 180,E1 -7014.14,E2 -7014.14} C_VEL
LIN {X 0,Y 481.93,Z 383.077,A -85,B 0,C 180,E1 -7017.493,E2 -7017.493} C_VEL
LIN {X 0,Y 481.907,Z 383.08,A -85,B 0,C 180,E1 -7020.836,E2 -7020.836} C_VEL
LIN {X 0,Y 481.929,Z 383.077,A -85,B 0,C 180,E1 -7022.508,E2 -7022.508} C_VEL
LIN {X 0,Y 481.818,Z 383.091,A -85,B 0,C 180,E1 -7025.86,E2 -7025.86} C_VEL
LIN {X 0,Y 481.765,Z 383.1,A -85,B 0,C 180,E1 -7028.388,E2 -7028.388} C_VEL
LIN {X 0,Y 481.753,Z 383.1,A -85,B 0,C 180,E1 -7031.785,E2 -7031.785} C_VEL
LIN {X 0,Y 481.746,Z 383.1,A -85,B 0,C 180,E1 -7035.224,E2 -7035.224} C_VEL
LIN {X 0,Y 481.715,Z 383.104,A -85,B 0,C 180,E1 -7038.722,E2 -7038.722} C_VEL
LIN {X 0,Y 481.65,Z 383.114,A -85,B 0,C 180,E1 -7041.395,E2 -7041.395} C_VEL
LIN {X 0,Y 481.68,Z 383.111,A -85,B 0,C 180,E1 -7044.113,E2 -7044.113} C_VEL
LIN {X 0,Y 481.749,Z 383.101,A -85,B 0,C 180,E1 -7047.139,E2 -7047.139} C_VEL
LIN {X 0,Y 481.681,Z 383.109,A -85,B 0,C 180,E1 -7049.741,E2 -7049.741} C_VEL
LIN {X 0,Y 481.674,Z 383.113,A -85,B 0,C 180,E1 -7052.674,E2 -7052.674} C_VEL
LIN {X 0,Y 481.646,Z 383.118,A -85,B 0,C 180,E1 -7055.709,E2 -7055.709} C_VEL
LIN {X 0,Y 481.674,Z 383.113,A -85,B 0,C 180,E1 -7058.859,E2 -7058.859} C_VEL
LIN {X 0,Y 481.655,Z 383.114,A -85,B 0,C 180,E1 -7061.913,E2 -7061.913} C_VEL
LIN {X 0,Y 481.661,Z 383.112,A -85,B 0,C 180,E1 -7064.457,E2 -7064.457} C_VEL
LIN {X 0,Y 481.685,Z 383.113,A -85,B 0,C 180,E1 -7066.847,E2 -7066.847} C_VEL
LIN {X 0,Y 481.659,Z 383.116,A -85,B 0,C 180,E1 -7070.058,E2 -7070.058} C_VEL
LIN {X 0,Y 481.849,Z 386.216,A -85,B 0,C 180,E1 -7072.223,E2 -7072.223} C_VEL
LIN {X 0,Y 481.755,Z 390.954,A -85,B 0,C 180,E1 -7075.323,E2 -7075.323} C_VEL
LIN {X 0,Y 481.605,Z 395.702,A -85,B 0,C 180,E1 -7078.309,E2 -7078.309} C_VEL
LIN {X 0,Y 481.441,Z 400.443,A -85,B 0,C 180,E1 -7081.202,E2 -7081.202} C_VEL
LIN {X 0,Y 481.312,Z 405.168,A -85,B 0,C 180,E1 -7084.02,E2 -7084.02} C_VEL
LIN {X 0,Y 481.209,Z 410.184,A -85,B 0,C 180,E1 -7086.942,E2 -7086.942} C_VEL
LIN {X 0,Y 481.178,Z 411.285,A -85,B 0,C 180,E1 -7087.575,E2 -7087.575} C_VEL
LIN {X 0,Y 480.505,Z 412.535,A -85,B 0,C 180,E1 -7088.257,E2 -7088.257} C_VEL
LIN {X 0,Y 477.604,Z 414.717,A -85,B 0,C 180,E1 -7089.36,E2 -7089.36} C_VEL
LIN {X 0,Y 475.138,Z 416.479,A -85,B 0,C 180,E1 -7090.249,E2 -7090.249} C_VEL
LIN {X 0,Y 474.068,Z 417.772,A -85,B 0,C 180,E1 -7090.937,E2 -7090.937} C_VEL
LIN {X 0,Y 473.975,Z 418.189,A -85,B 0,C 180,E1 -7091.171,E2 -7091.171} C_VEL
LIN {X 0,Y 473.975,Z 419.128,A -85,B 0,C 180,E1 -7091.705,E2 -7091.705} C_VEL
LIN {X 0,Y 477.64,Z 434.681,A -85,B 0,C 180,E1 -7092.237,E2 -7092.237} C_VEL
LIN {X 0,Y 478.6,Z 439.996,A -85,B 0,C 180,E1 -7092.453,E2 -7092.453} C_VEL
LIN {X 0,Y 478.176,Z 452.628,A -85,B 0,C 180,E1 -7092.968,E2 -7092.968} C_VEL
LIN {X 0,Y 477.686,Z 465.518,A -85,B 0,C 180,E1 -7093.661,E2 -7093.661} C_VEL
LIN {X 0,Y 477.075,Z 478.058,A -85,B 0,C 180,E1 -7094.514,E2 -7094.514} C_VEL
LIN {X 0,Y 476.424,Z 489.525,A -85,B 0,C 180,E1 -7095.477,E2 -7095.477} C_VEL
LIN {X 0,Y 475.79,Z 500.048,A -85,B 0,C 180,E1 -7096.547,E2 -7096.547} C_VEL
LIN {X 0,Y 475.285,Z 510.259,A -85,B 0,C 180,E1 -7097.805,E2 -7097.805} C_VEL
LIN {X 0,Y 474.784,Z 519.109,A -85,B 0,C 180,E1 -7099.121,E2 -7099.121} C_VEL
LIN {X 0,Y 474.364,Z 527.37,A -85,B 0,C 180,E1 -7100.621,E2 -7100.621} C_VEL
LIN {X 0,Y 474.113,Z 533.124,A -85,B 0,C 180,E1 -7101.905,E2 -7101.905} C_VEL
LIN {X 0,Y 473.955,Z 538.786,A -85,B 0,C 180,E1 -7103.467,E2 -7103.467} C_VEL
LIN {X 0,Y 473.838,Z 542.761,A -85,B 0,C 180,E1 -7104.894,E2 -7104.894} C_VEL
LIN {X 0,Y 473.792,Z 546.176,A -85,B 0,C 180,E1 -7106.598,E2 -7106.598} C_VEL
LIN {X 0,Y 473.697,Z 548.207,A -85,B 0,C 180,E1 -7108.3,E2 -7108.3} C_VEL
LIN {X 0,Y 473.668,Z 548.907,A -85,B 0,C 180,E1 -7110,E2 -7110} C_VEL
LIN {X 0,Y 473.696,Z 548.285,A -85,B 0,C 180,E1 -7111.7,E2 -7111.7} C_VEL
LIN {X 0,Y 473.791,Z 546.324,A -85,B 0,C 180,E1 -7113.402,E2 -7113.402} C_VEL
LIN {X 0,Y 473.835,Z 542.981,A -85,B 0,C 180,E1 -7115.106,E2 -7115.106} C_VEL
LIN {X 0,Y 473.929,Z 538.158,A -85,B 0,C 180,E1 -7116.813,E2 -7116.813} C_VEL
LIN {X 0,Y 474.199,Z 531.698,A -85,B 0,C 180,E1 -7118.523,E2 -7118.523} C_VEL
LIN {X 0,Y 474.495,Z 524.506,A -85,B 0,C 180,E1 -7120.023,E2 -7120.023} C_VEL
LIN {X 0,Y 475.003,Z 515.61,A -85,B 0,C 180,E1 -7121.522,E2 -7121.522} C_VEL
LIN {X 0,Y 475.499,Z 506.265,A -85,B 0,C 180,E1 -7122.809,E2 -7122.809} C_VEL
LIN {X 0,Y 476.057,Z 495.915,A -85,B 0,C 180,E1 -7123.99,E2 -7123.99} C_VEL
LIN {X 0,Y 476.699,Z 484.493,A -85,B 0,C 180,E1 -7125.061,E2 -7125.061} C_VEL
LIN {X 0,Y 477.379,Z 471.834,A -85,B 0,C 180,E1 -7126.024,E2 -7126.024} C_VEL
LIN {X 0,Y 477.906,Z 459.955,A -85,B 0,C 180,E1 -7126.751,E2 -7126.751} C_VEL
LIN {X 0,Y 478.418,Z 445.898,A -85,B 0,C 180,E1 -7127.416,E2 -7127.416} C_VEL
LIN {X 0,Y 478.46,Z 438.882,A -85,B 0,C 180,E1 -7127.683,E2 -7127.683} C_VEL
LIN {X 0,Y 475.362,Z 424.9,A -85,B 0,C 180,E1 -7128.207,E2 -7128.207} C_VEL
LIN {X 0,Y 473.971,Z 419.098,A -85,B 0,C 180,E1 -7128.403,E2 -7128.403} C_VEL
LIN {X 0,Y 474.078,Z 413.261,A -85,B 0,C 180,E1 -7131.754,E2 -7131.754} C_VEL
LIN {X 0,Y 474.188,Z 408.53,A -85,B 0,C 180,E1 -7134.519,E2 -7134.519} C_VEL
LIN {X 0,Y 474.304,Z 403.802,A -85,B 0,C 180,E1 -7137.345,E2 -7137.345} C_VEL
LIN {X 0,Y 474.523,Z 398.166,A -85,B 0,C 180,E1 -7140.793,E2 -7140.793} C_VEL
LIN {X 0,Y 474.642,Z 394.304,A -85,B 0,C 180,E1 -7143.22,E2 -7143.22} C_VEL
LIN {X 0,Y 474.758,Z 389.553,A -85,B 0,C 180,E1 -7146.309,E2 -7146.309} C_VEL
LIN {X 0,Y 474.777,Z 386.393,A -85,B 0,C 180,E1 -7148.442,E2 -7148.442} C_VEL
LIN {X 0,Y 474.711,Z 384.637,A -85,B 0,C 180,E1 -7149.659,E2 -7149.659} C_VEL
LIN {X 0,Y 474.635,Z 383.993,A -85,B 0,C 180,E1 -7150.96,E2 -7150.96} C_VEL
LIN {X 0,Y 474.618,Z 383.991,A -85,B 0,C 180,E1 -7154.104,E2 -7154.104} C_VEL
LIN {X 0,Y 474.618,Z 383.991,A -85,B 0,C 180,E1 -7157.066,E2 -7157.066} C_VEL
LIN {X 0,Y 474.647,Z 383.985,A -85,B 0,C 180,E1 -7160.454,E2 -7160.454} C_VEL
LIN {X 0,Y 474.596,Z 383.991,A -85,B 0,C 180,E1 -7163.677,E2 -7163.677} C_VEL
LIN {X 0,Y 474.646,Z 383.985,A -85,B 0,C 180,E1 -7166.78,E2 -7166.78} C_VEL
LIN {X 0,Y 474.608,Z 383.99,A -85,B 0,C 180,E1 -7169.77,E2 -7169.77} C_VEL
LIN {X 0,Y 474.7,Z 383.981,A -85,B 0,C 180,E1 -7172.68,E2 -7172.68} C_VEL
LIN {X 0,Y 474.66,Z 383.986,A -85,B 0,C 180,E1 -7175.507,E2 -7175.507} C_VEL
LIN {X 0,Y 474.674,Z 383.982,A -85,B 0,C 180,E1 -7179.185,E2 -7179.185} C_VEL
LIN {X 0,Y 474.659,Z 383.985,A -85,B 0,C 180,E1 -7181.884,E2 -7181.884} C_VEL
LIN {X 0,Y 474.704,Z 383.977,A -85,B 0,C 180,E1 -7184.544,E2 -7184.544} C_VEL
LIN {X 0,Y 474.708,Z 383.977,A -85,B 0,C 180,E1 -7188.038,E2 -7188.038} C_VEL
LIN {X 0,Y 474.731,Z 383.974,A -85,B 0,C 180,E1 -7191.486,E2 -7191.486} C_VEL
LIN {X 0,Y 474.782,Z 383.968,A -85,B 0,C 180,E1 -7194.052,E2 -7194.052} C_VEL
LIN {X 0,Y 474.897,Z 383.953,A -85,B 0,C 180,E1 -7197.455,E2 -7197.455} C_VEL
LIN {X 0,Y 474.915,Z 383.956,A -85,B 0,C 180,E1 -7200,E2 -7200} C_VEL
LIN {X 0,Y 474.897,Z 383.953,A -85,B 0,C 180,E1 -7202.545,E2 -7202.545} C_VEL
LIN {X 0,Y 474.782,Z 383.967,A -85,B 0,C 180,E1 -7205.947,E2 -7205.947} C_VEL
LIN {X 0,Y 474.73,Z 383.976,A -85,B 0,C 180,E1 -7208.513,E2 -7208.513} C_VEL
LIN {X 0,Y 474.708,Z 383.977,A -85,B 0,C 180,E1 -7211.962,E2 -7211.962} C_VEL
LIN {X 0,Y 474.704,Z 383.977,A -85,B 0,C 180,E1 -7215.455,E2 -7215.455} C_VEL
LIN {X 0,Y 474.669,Z 383.983,A -85,B 0,C 180,E1 -7219.01,E2 -7219.01} C_VEL
LIN {X 0,Y 474.593,Z 383.992,A -85,B 0,C 180,E1 -7221.729,E2 -7221.729} C_VEL
LIN {X 0,Y 474.662,Z 383.986,A -85,B 0,C 180,E1 -7224.493,E2 -7224.493} C_VEL
LIN {X 0,Y 474.702,Z 383.979,A -85,B 0,C 180,E1 -7227.339,E2 -7227.339} C_VEL
LIN {X 0,Y 474.607,Z 383.993,A -85,B 0,C 180,E1 -7230.81,E2 -7230.81} C_VEL
LIN {X 0,Y 474.641,Z 383.991,A -85,B 0,C 180,E1 -7233.984,E2 -7233.984} C_VEL
LIN {X 0,Y 474.579,Z 383.996,A -85,B 0,C 180,E1 -7236.9,E2 -7236.9} C_VEL
LIN {X 0,Y 474.657,Z 383.986,A -85,B 0,C 180,E1 -7239.652,E2 -7239.652} C_VEL
LIN {X 0,Y 474.616,Z 383.99,A -85,B 0,C 180,E1 -7242.934,E2 -7242.934} C_VEL
LIN {X 0,Y 474.608,Z 383.993,A -85,B 0,C 180,E1 -7245.895,E2 -7245.895} C_VEL
LIN {X 0,Y 474.672,Z 384.118,A -85,B 0,C 180,E1 -7248.768,E2 -7248.768} C_VEL
LIN {X 0,Y 475.036,Z 386.917,A -85,B 0,C 180,E1 -7250.493,E2 -7250.493} C_VEL
LIN {X 0,Y 475.142,Z 391.2,A -85,B 0,C 180,E1 -7253.009,E2 -7253.009} C_VEL
LIN {X 0,Y 474.918,Z 396.493,A -85,B 0,C 180,E1 -7255.966,E2 -7255.966} C_VEL
LIN {X 0,Y 474.667,Z 402.432,A -85,B 0,C 180,E1 -7259.177,E2 -7259.177} C_VEL
LIN {X 0,Y 474.458,Z 409.206,A -85,B 0,C 180,E1 -7262.718,E2 -7262.718} C_VEL
LIN {X 0,Y 474.283,Z 414.677,A -85,B 0,C 180,E1 -7265.486,E2 -7265.486} C_VEL
LIN {X 0,Y 474.165,Z 421.841,A -85,B 0,C 180,E1 -7269.031,E2 -7269.031} C_VEL
LIN {X 0,Y 474.035,Z 427.265,A -85,B 0,C 180,E1 -7271.659,E2 -7271.659} C_VEL
LIN {X 0,Y 477.335,Z 442.361,A -85,B 0,C 180,E1 -7272.145,E2 -7272.145} C_VEL
LIN {X 0,Y 478.562,Z 449.343,A -85,B 0,C 180,E1 -7272.424,E2 -7272.424} C_VEL
LIN {X 0,Y 478.123,Z 462.185,A -85,B 0,C 180,E1 -7272.954,E2 -7272.954} C_VEL
LIN {X 0,Y 477.543,Z 475.206,A -85,B 0,C 180,E1 -7273.66,E2 -7273.66} C_VEL
LIN {X 0,Y 476.907,Z 487.557,A -85,B 0,C 180,E1 -7274.508,E2 -7274.508} C_VEL
LIN {X 0,Y 476.306,Z 498.954,A -85,B 0,C 180,E1 -7275.473,E2 -7275.473} C_VEL
LIN {X 0,Y 475.688,Z 509.426,A -85,B 0,C 180,E1 -7276.544,E2 -7276.544} C_VEL
LIN {X 0,Y 475.154,Z 519.757,A -85,B 0,C 180,E1 -7277.821,E2 -7277.821} C_VEL
LIN {X 0,Y 474.718,Z 528.435,A -85,B 0,C 180,E1 -7279.12,E2 -7279.12} C_VEL
LIN {X 0,Y 474.306,Z 536.662,A -85,B 0,C 180,E1 -7280.619,E2 -7280.619} C_VEL
LIN {X 0,Y 474.067,Z 542.42,A -85,B 0,C 180,E1 -7281.904,E2 -7281.904} C_VEL
LIN {X 0,Y 473.882,Z 548.323,A -85,B 0,C 180,E1 -7283.544,E2 -7283.544} C_VEL
LIN {X 0,Y 473.831,Z 552.026,A -85,B 0,C 180,E1 -7284.894,E2 -7284.894} C_VEL
LIN {X 0,Y 473.755,Z 555.424,A -85,B 0,C 180,E1 -7286.598,E2 -7286.598} C_VEL
LIN {X 0,Y 473.692,Z 557.433,A -85,B 0,C 180,E1 -7288.3,E2 -7288.3} C_VEL
LIN {X 0,Y 473.668,Z 558.1,A -85,B 0,C 180,E1 -7290,E2 -7290} C_VEL
LIN {X 0,Y 473.692,Z 557.435,A -85,B 0,C 180,E1 -7291.7,E2 -7291.7} C_VEL
LIN {X 0,Y 473.755,Z 555.428,A -85,B 0,C 180,E1 -7293.402,E2 -7293.402} C_VEL
LIN {X 0,Y 473.83,Z 552.029,A -85,B 0,C 180,E1 -7295.106,E2 -7295.106} C_VEL
LIN {X 0,Y 473.912,Z 547.137,A -85,B 0,C 180,E1 -7296.813,E2 -7296.813} C_VEL
LIN {X 0,Y 474.139,Z 540.607,A -85,B 0,C 180,E1 -7298.524,E2 -7298.524} C_VEL
LIN {X 0,Y 474.452,Z 533.34,A -85,B 0,C 180,E1 -7300.023,E2 -7300.023} C_VEL
LIN {X 0,Y 474.955,Z 524.341,A -85,B 0,C 180,E1 -7301.523,E2 -7301.523} C_VEL
LIN {X 0,Y 475.401,Z 514.894,A -85,B 0,C 180,E1 -7302.812,E2 -7302.812} C_VEL
LIN {X 0,Y 475.955,Z 504.435,A -85,B 0,C 180,E1 -7303.992,E2 -7303.992} C_VEL
LIN {X 0,Y 476.595,Z 492.894,A -85,B 0,C 180,E1 -7305.064,E2 -7305.064} C_VEL
LIN {X 0,Y 477.317,Z 480.091,A -85,B 0,C 180,E1 -7306.026,E2 -7306.026} C_VEL
LIN {X 0,Y 477.843,Z 468.369,A -85,B 0,C 180,E1 -7306.733,E2 -7306.733} C_VEL
LIN {X 0,Y 478.325,Z 454.979,A -85,B 0,C 180,E1 -7307.364,E2 -7307.364} C_VEL
LIN {X 0,Y 478.359,Z 447.797,A -85,B 0,C 180,E1 -7307.639,E2 -7307.639} C_VEL
LIN {X 0,Y 475.535,Z 433.841,A -85,B 0,C 180,E1 -7308.15,E2 -7308.15} C_VEL
LIN {X 0,Y 474.041,Z 427.216,A -85,B 0,C 180,E1 -7308.364,E2 -7308.364} C_VEL
LIN {X 0,Y 474.159,Z 420.244,A -85,B 0,C 180,E1 -7311.75,E2 -7311.75} C_VEL
LIN {X 0,Y 474.283,Z 414.674,A -85,B 0,C 180,E1 -7314.514,E2 -7314.514} C_VEL
LIN {X 0,Y 474.458,Z 409.098,A -85,B 0,C 180,E1 -7317.335,E2 -7317.335} C_VEL
LIN {X 0,Y 474.665,Z 402.42,A -85,B 0,C 180,E1 -7320.822,E2 -7320.822} C_VEL
LIN {X 0,Y 474.917,Z 396.483,A -85,B 0,C 180,E1 -7324.034,E2 -7324.034} C_VEL
LIN {X 0,Y 475.142,Z 391.193,A -85,B 0,C 180,E1 -7326.991,E2 -7326.991} C_VEL
LIN {X 0,Y 475.038,Z 386.906,A -85,B 0,C 180,E1 -7329.507,E2 -7329.507} C_VEL
LIN {X 0,Y 474.636,Z 383.993,A -85,B 0,C 180,E1 -7331.345,E2 -7331.345} C_VEL
LIN {X 0,Y 474.617,Z 383.994,A -85,B 0,C 180,E1 -7334.702,E2 -7334.702} C_VEL
LIN {X 0,Y 474.627,Z 383.993,A -85,B 0,C 180,E1 -7337.763,E2 -7337.763} C_VEL
LIN {X 0,Y 474.675,Z 383.982,A -85,B 0,C 180,E1 -7340.457,E2 -7340.457} C_VEL
LIN {X 0,Y 474.596,Z 383.992,A -85,B 0,C 180,E1 -7343.677,E2 -7343.677} C_VEL
LIN {X 0,Y 474.644,Z 383.986,A -85,B 0,C 180,E1 -7346.78,E2 -7346.78} C_VEL
LIN {X 0,Y 474.607,Z 383.991,A -85,B 0,C 180,E1 -7349.77,E2 -7349.77} C_VEL
LIN {X 0,Y 474.698,Z 383.981,A -85,B 0,C 180,E1 -7352.68,E2 -7352.68} C_VEL
LIN {X 0,Y 474.64,Z 383.989,A -85,B 0,C 180,E1 -7355.506,E2 -7355.506} C_VEL
LIN {X 0,Y 474.672,Z 383.984,A -85,B 0,C 180,E1 -7359.185,E2 -7359.185} C_VEL
LIN {X 0,Y 474.659,Z 383.985,A -85,B 0,C 180,E1 -7361.884,E2 -7361.884} C_VEL
LIN {X 0,Y 474.703,Z 383.977,A -85,B 0,C 180,E1 -7364.544,E2 -7364.544} C_VEL
LIN {X 0,Y 474.706,Z 383.977,A -85,B 0,C 180,E1 -7368.038,E2 -7368.038} C_VEL
LIN {X 0,Y 474.73,Z 383.975,A -85,B 0,C 180,E1 -7371.487,E2 -7371.487} C_VEL
LIN {X 0,Y 474.781,Z 383.968,A -85,B 0,C 180,E1 -7374.052,E2 -7374.052} C_VEL
LIN {X 0,Y 474.896,Z 383.953,A -85,B 0,C 180,E1 -7377.455,E2 -7377.455} C_VEL
LIN {X 0,Y 474.914,Z 383.956,A -85,B 0,C 180,E1 -7380,E2 -7380} C_VEL
LIN {X 0,Y 474.895,Z 383.953,A -85,B 0,C 180,E1 -7382.545,E2 -7382.545} C_VEL
LIN {X 0,Y 474.781,Z 383.968,A -85,B 0,C 180,E1 -7385.948,E2 -7385.948} C_VEL
LIN {X 0,Y 474.73,Z 383.975,A -85,B 0,C 180,E1 -7388.514,E2 -7388.514} C_VEL
LIN {X 0,Y 474.706,Z 383.977,A -85,B 0,C 180,E1 -7391.962,E2 -7391.962} C_VEL
LIN {X 0,Y 474.703,Z 383.977,A -85,B 0,C 180,E1 -7395.456,E2 -7395.456} C_VEL
LIN {X 0,Y 474.668,Z 383.983,A -85,B 0,C 180,E1 -7399.01,E2 -7399.01} C_VEL
LIN {X 0,Y 474.592,Z 383.991,A -85,B 0,C 180,E1 -7401.729,E2 -7401.729} C_VEL
LIN {X 0,Y 474.662,Z 383.987,A -85,B 0,C 180,E1 -7404.493,E2 -7404.493} C_VEL
LIN {X 0,Y 474.701,Z 383.98,A -85,B 0,C 180,E1 -7407.339,E2 -7407.339} C_VEL
LIN {X 0,Y 474.606,Z 383.995,A -85,B 0,C 180,E1 -7410.81,E2 -7410.81} C_VEL
LIN {X 0,Y 474.641,Z 383.99,A -85,B 0,C 180,E1 -7413.984,E2 -7413.984} C_VEL
LIN {X 0,Y 474.579,Z 383.995,A -85,B 0,C 180,E1 -7416.9,E2 -7416.9} C_VEL
LIN {X 0,Y 474.63,Z 383.987,A -85,B 0,C 180,E1 -7419.648,E2 -7419.648} C_VEL
LIN {X 0,Y 474.617,Z 383.989,A -85,B 0,C 180,E1 -7422.934,E2 -7422.934} C_VEL
LIN {X 0,Y 474.62,Z 383.991,A -85,B 0,C 180,E1 -7425.896,E2 -7425.896} C_VEL
LIN {X 0,Y 474.634,Z 383.991,A -85,B 0,C 180,E1 -7429.04,E2 -7429.04} C_VEL
LIN {X 0,Y 474.672,Z 384.668,A -85,B 0,C 180,E1 -7430.457,E2 -7430.457} C_VEL
LIN {X 0,Y 474.798,Z 388.468,A -85,B 0,C 180,E1 -7433.065,E2 -7433.065} C_VEL
LIN {X 0,Y 474.702,Z 392.942,A -85,B 0,C 180,E1 -7436.005,E2 -7436.005} C_VEL
LIN {X 0,Y 474.519,Z 397.326,A -85,B 0,C 180,E1 -7438.777,E2 -7438.777} C_VEL
LIN {X 0,Y 474.361,Z 402.069,A -85,B 0,C 180,E1 -7441.699,E2 -7441.699} C_VEL
LIN {X 0,Y 474.252,Z 407.036,A -85,B 0,C 180,E1 -7444.685,E2 -7444.685} C_VEL
LIN {X 0,Y 474.099,Z 411.912,A -85,B 0,C 180,E1 -7447.555,E2 -7447.555} C_VEL
LIN {X 0,Y 473.995,Z 416.251,A -85,B 0,C 180,E1 -7450.061,E2 -7450.061} C_VEL
LIN {X 0,Y 473.975,Z 418.189,A -85,B 0,C 180,E1 -7451.171,E2 -7451.171} C_VEL
LIN {X 0,Y 473.95,Z 419.503,A -85,B 0,C 180,E1 -7451.446,E2 -7451.446} C_VEL
LIN {X 0,Y 473.889,Z 422.43,A -85,B 0,C 180,E1 -7451.681,E2 -7451.681} C_VEL
LIN {X 0,Y 473.656,Z 429.037,A -85,B 0,C 180,E1 -7451.917,E2 -7451.917} C_VEL
LIN {X 0,Y 472.075,Z 442.885,A -85,B 0,C 180,E1 -7452.296,E2 -7452.296} C_VEL
LIN {X 0,Y 471.556,Z 447.954,A -85,B 0,C 180,E1 -7452.5,E2 -7452.5} C_VEL
LIN {X 0,Y 471.095,Z 460.525,A -85,B 0,C 180,E1 -7453.12,E2 -7453.12} C_VEL
LIN {X 0,Y 470.474,Z 473.776,A -85,B 0,C 180,E1 -7453.957,E2 -7453.957} C_VEL
LIN {X 0,Y 469.684,Z 486.076,A -85,B 0,C 180,E1 -7454.931,E2 -7454.931} C_VEL
LIN {X 0,Y 469.034,Z 497.201,A -85,B 0,C 180,E1 -7456.018,E2 -7456.018} C_VEL
LIN {X 0,Y 468.471,Z 507.171,A -85,B 0,C 180,E1 -7457.196,E2 -7457.196} C_VEL
LIN {X 0,Y 468.01,Z 516.48,A -85,B 0,C 180,E1 -7458.523,E2 -7458.523} C_VEL
LIN {X 0,Y 467.509,Z 524.115,A -85,B 0,C 180,E1 -7459.826,E2 -7459.826} C_VEL
LIN {X 0,Y 467.147,Z 531.392,A -85,B 0,C 180,E1 -7461.347,E2 -7461.347} C_VEL
LIN {X 0,Y 466.901,Z 537.929,A -85,B 0,C 180,E1 -7463.084,E2 -7463.084} C_VEL
LIN {X 0,Y 466.776,Z 542.831,A -85,B 0,C 180,E1 -7464.817,E2 -7464.817} C_VEL
LIN {X 0,Y 466.688,Z 546.246,A -85,B 0,C 180,E1 -7466.547,E2 -7466.547} C_VEL
LIN {X 0,Y 466.606,Z 548.276,A -85,B 0,C 180,E1 -7468.274,E2 -7468.274} C_VEL
LIN {X 0,Y 466.597,Z 548.976,A -85,B 0,C 180,E1 -7470,E2 -7470} C_VEL
LIN {X 0,Y 466.605,Z 548.353,A -85,B 0,C 180,E1 -7471.726,E2 -7471.726} C_VEL
LIN {X 0,Y 466.687,Z 546.392,A -85,B 0,C 180,E1 -7473.454,E2 -7473.454} C_VEL
LIN {X 0,Y 466.771,Z 543.048,A -85,B 0,C 180,E1 -7475.183,E2 -7475.183} C_VEL
LIN {X 0,Y 466.852,Z 538.224,A -85,B 0,C 180,E1 -7476.917,E2 -7476.917} C_VEL
LIN {X 0,Y 467.134,Z 531.765,A -85,B 0,C 180,E1 -7478.653,E2 -7478.653} C_VEL
LIN {X 0,Y 467.461,Z 524.572,A -85,B 0,C 180,E1 -7480.175,E2 -7480.175} C_VEL
LIN {X 0,Y 468.019,Z 515.676,A -85,B 0,C 180,E1 -7481.696,E2 -7481.696} C_VEL
LIN {X 0,Y 468.534,Z 506.33,A -85,B 0,C 180,E1 -7483.003,E2 -7483.003} C_VEL
LIN {X 0,Y 469.154,Z 495.978,A -85,B 0,C 180,E1 -7484.2,E2 -7484.2} C_VEL
LIN {X 0,Y 469.811,Z 484.556,A -85,B 0,C 180,E1 -7485.287,E2 -7485.287} C_VEL
LIN {X 0,Y 470.548,Z 471.896,A -85,B 0,C 180,E1 -7486.263,E2 -7486.263} C_VEL
LIN {X 0,Y 471.181,Z 458.692,A -85,B 0,C 180,E1 -7487.071,E2 -7487.071} C_VEL
LIN {X 0,Y 471.697,Z 444.655,A -85,B 0,C 180,E1 -7487.728,E2 -7487.728} C_VEL
LIN {X 0,Y 471.705,Z 440.266,A -85,B 0,C 180,E1 -7487.896,E2 -7487.896} C_VEL
LIN {X 0,Y 468.722,Z 426.551,A -85,B 0,C 180,E1 -7488.434,E2 -7488.434} C_VEL
LIN {X 0,Y 466.913,Z 419.188,A -85,B 0,C 180,E1 -7488.677,E2 -7488.677} C_VEL
LIN {X 0,Y 467.004,Z 413.316,A -85,B 0,C 180,E1 -7492.1,E2 -7492.1} C_VEL
LIN {X 0,Y 467.155,Z 408.589,A -85,B 0,C 180,E1 -7494.913,E2 -7494.913} C_VEL
LIN {X 0,Y 467.256,Z 403.846,A -85,B 0,C 180,E1 -7497.793,E2 -7497.793} C_VEL
LIN {X 0,Y 467.48,Z 398.653,A -85,B 0,C 180,E1 -7501.026,E2 -7501.026} C_VEL
LIN {X 0,Y 467.61,Z 394.343,A -85,B 0,C 180,E1 -7503.786,E2 -7503.786} C_VEL
LIN {X 0,Y 467.764,Z 389.591,A -85,B 0,C 180,E1 -7506.941,E2 -7506.941} C_VEL
LIN {X 0,Y 467.634,Z 385.259,A -85,B 0,C 180,E1 -7509.962,E2 -7509.962} C_VEL
LIN {X 0,Y 467.586,Z 384.872,A -85,B 0,C 180,E1 -7510.264,E2 -7510.264} C_VEL
LIN {X 0,Y 467.589,Z 384.867,A -85,B 0,C 180,E1 -7512.567,E2 -7512.567} C_VEL
LIN {X 0,Y 467.573,Z 384.869,A -85,B 0,C 180,E1 -7515.053,E2 -7515.053} C_VEL
LIN {X 0,Y 467.591,Z 384.867,A -85,B 0,C 180,E1 -7517.44,E2 -7517.44} C_VEL
LIN {X 0,Y 467.585,Z 384.868,A -85,B 0,C 180,E1 -7520.855,E2 -7520.855} C_VEL
LIN {X 0,Y 467.566,Z 384.87,A -85,B 0,C 180,E1 -7524.26,E2 -7524.26} C_VEL
LIN {X 0,Y 467.585,Z 384.867,A -85,B 0,C 180,E1 -7527.321,E2 -7527.321} C_VEL
LIN {X 0,Y 467.573,Z 384.868,A -85,B 0,C 180,E1 -7530.667,E2 -7530.667} C_VEL
LIN {X 0,Y 467.619,Z 384.86,A -85,B 0,C 180,E1 -7533.2,E2 -7533.2} C_VEL
LIN {X 0,Y 467.596,Z 384.861,A -85,B 0,C 180,E1 -7536.468,E2 -7536.468} C_VEL
LIN {X 0,Y 467.626,Z 384.857,A -85,B 0,C 180,E1 -7539.777,E2 -7539.777} C_VEL
LIN {X 0,Y 467.61,Z 384.863,A -85,B 0,C 180,E1 -7542.507,E2 -7542.507} C_VEL
LIN {X 0,Y 467.613,Z 384.863,A -85,B 0,C 180,E1 -7545.197,E2 -7545.197} C_VEL
LIN {X 0,Y 467.659,Z 384.855,A -85,B 0,C 180,E1 -7547.855,E2 -7547.855} C_VEL
LIN {X 0,Y 467.685,Z 384.851,A -85,B 0,C 180,E1 -7551.357,E2 -7551.357} C_VEL
LIN {X 0,Y 467.747,Z 384.845,A -85,B 0,C 180,E1 -7553.963,E2 -7553.963} C_VEL
LIN {X 0,Y 467.862,Z 384.83,A -85,B 0,C 180,E1 -7557.417,E2 -7557.417} C_VEL
LIN {X 0,Y 467.885,Z 384.832,A -85,B 0,C 180,E1 -7560,E2 -7560} C_VEL
LIN {X 0,Y 467.863,Z 384.83,A -85,B 0,C 180,E1 -7562.583,E2 -7562.583} C_VEL
LIN {X 0,Y 467.747,Z 384.844,A -85,B 0,C 180,E1 -7566.037,E2 -7566.037} C_VEL
LIN {X 0,Y 467.684,Z 384.853,A -85,B 0,C 180,E1 -7568.643,E2 -7568.643} C_VEL
LIN {X 0,Y 467.659,Z 384.855,A -85,B 0,C 180,E1 -7572.145,E2 -7572.145} C_VEL
LIN {X 0,Y 467.643,Z 384.858,A -85,B 0,C 180,E1 -7575.695,E2 -7575.695} C_VEL
LIN {X 0,Y 467.621,Z 384.86,A -85,B 0,C 180,E1 -7578.765,E2 -7578.765} C_VEL
LIN {X 0,Y 467.584,Z 384.868,A -85,B 0,C 180,E1 -7581.268,E2 -7581.268} C_VEL
LIN {X 0,Y 467.576,Z 384.865,A -85,B 0,C 180,E1 -7583.943,E2 -7583.943} C_VEL
LIN {X 0,Y 467.619,Z 384.859,A -85,B 0,C 180,E1 -7586.8,E2 -7586.8} C_VEL
LIN {X 0,Y 467.557,Z 384.867,A -85,B 0,C 180,E1 -7589.738,E2 -7589.738} C_VEL
LIN {X 0,Y 467.585,Z 384.867,A -85,B 0,C 180,E1 -7592.758,E2 -7592.758} C_VEL
LIN {X 0,Y 467.559,Z 384.873,A -85,B 0,C 180,E1 -7595.889,E2 -7595.889} C_VEL
LIN {X 0,Y 467.621,Z 384.865,A -85,B 0,C 180,E1 -7599.141,E2 -7599.141} C_VEL
LIN {X 0,Y 467.588,Z 384.867,A -85,B 0,C 180,E1 -7602.567,E2 -7602.567} C_VEL
LIN {X 0,Y 467.568,Z 384.87,A -85,B 0,C 180,E1 -7605.052,E2 -7605.052} C_VEL
LIN {X 0,Y 467.605,Z 384.927,A -85,B 0,C 180,E1 -7608.528,E2 -7608.528} C_VEL
LIN {X 0,Y 468.069,Z 388.73,A -85,B 0,C 180,E1 -7610.903,E2 -7610.903} C_VEL
LIN {X 0,Y 468.107,Z 392.419,A -85,B 0,C 180,E1 -7613.091,E2 -7613.091} C_VEL
LIN {X 0,Y 467.868,Z 397.969,A -85,B 0,C 180,E1 -7616.235,E2 -7616.235} C_VEL
LIN {X 0,Y 467.621,Z 403.504,A -85,B 0,C 180,E1 -7619.27,E2 -7619.27} C_VEL
LIN {X 0,Y 467.408,Z 409.625,A -85,B 0,C 180,E1 -7622.515,E2 -7622.515} C_VEL
LIN {X 0,Y 467.237,Z 414.619,A -85,B 0,C 180,E1 -7625.092,E2 -7625.092} C_VEL
LIN {X 0,Y 467.102,Z 420.187,A -85,B 0,C 180,E1 -7627.904,E2 -7627.904} C_VEL
LIN {X 0,Y 466.967,Z 426.923,A -85,B 0,C 180,E1 -7631.236,E2 -7631.236} C_VEL
LIN {X 0,Y 466.963,Z 427.191,A -85,B 0,C 180,E1 -7631.367,E2 -7631.367} C_VEL
LIN {X 0,Y 470.492,Z 443.021,A -85,B 0,C 180,E1 -7631.899,E2 -7631.899} C_VEL
LIN {X 0,Y 471.755,Z 450.336,A -85,B 0,C 180,E1 -7632.201,E2 -7632.201} C_VEL
LIN {X 0,Y 471.277,Z 463.163,A -85,B 0,C 180,E1 -7632.75,E2 -7632.75} C_VEL
LIN {X 0,Y 470.607,Z 476.784,A -85,B 0,C 180,E1 -7633.516,E2 -7633.516} C_VEL
LIN {X 0,Y 469.983,Z 488.916,A -85,B 0,C 180,E1 -7634.385,E2 -7634.385} C_VEL
LIN {X 0,Y 469.346,Z 500.06,A -85,B 0,C 180,E1 -7635.363,E2 -7635.363} C_VEL
LIN {X 0,Y 468.63,Z 511.256,A -85,B 0,C 180,E1 -7636.558,E2 -7636.558} C_VEL
LIN {X 0,Y 468.086,Z 521.295,A -85,B 0,C 180,E1 -7637.866,E2 -7637.866} C_VEL
LIN {X 0,Y 467.62,Z 529.633,A -85,B 0,C 180,E1 -7639.172,E2 -7639.172} C_VEL
LIN {X 0,Y 467.212,Z 537.603,A -85,B 0,C 180,E1 -7640.694,E2 -7640.694} C_VEL
LIN {X 0,Y 466.915,Z 544.02,A -85,B 0,C 180,E1 -7642.214,E2 -7642.214} C_VEL
LIN {X 0,Y 466.773,Z 549.708,A -85,B 0,C 180,E1 -7643.95,E2 -7643.95} C_VEL
LIN {X 0,Y 466.764,Z 551.957,A -85,B 0,C 180,E1 -7644.817,E2 -7644.817} C_VEL
LIN {X 0,Y 466.651,Z 555.354,A -85,B 0,C 180,E1 -7646.546,E2 -7646.546} C_VEL
LIN {X 0,Y 466.601,Z 557.364,A -85,B 0,C 180,E1 -7648.274,E2 -7648.274} C_VEL
LIN {X 0,Y 466.597,Z 558.031,A -85,B 0,C 180,E1 -7650,E2 -7650} C_VEL
LIN {X 0,Y 466.601,Z 557.366,A -85,B 0,C 180,E1 -7651.726,E2 -7651.726} C_VEL
LIN {X 0,Y 466.651,Z 555.359,A -85,B 0,C 180,E1 -7653.454,E2 -7653.454} C_VEL
LIN {X 0,Y 466.764,Z 551.961,A -85,B 0,C 180,E1 -7655.183,E2 -7655.183} C_VEL
LIN {X 0,Y 466.833,Z 547.068,A -85,B 0,C 180,E1 -7656.917,E2 -7656.917} C_VEL
LIN {X 0,Y 467.082,Z 540.538,A -85,B 0,C 180,E1 -7658.654,E2 -7658.654} C_VEL
LIN {X 0,Y 467.399,Z 533.27,A -85,B 0,C 180,E1 -7660.176,E2 -7660.176} C_VEL
LIN {X 0,Y 467.966,Z 524.271,A -85,B 0,C 180,E1 -7661.698,E2 -7661.698} C_VEL
LIN {X 0,Y 468.45,Z 514.823,A -85,B 0,C 180,E1 -7663.005,E2 -7663.005} C_VEL
LIN {X 0,Y 469.044,Z 504.365,A -85,B 0,C 180,E1 -7664.203,E2 -7664.203} C_VEL
LIN {X 0,Y 469.729,Z 492.824,A -85,B 0,C 180,E1 -7665.29,E2 -7665.29} C_VEL
LIN {X 0,Y 470.465,Z 480.019,A -85,B 0,C 180,E1 -7666.266,E2 -7666.266} C_VEL
LIN {X 0,Y 471.077,Z 467.133,A -85,B 0,C 180,E1 -7667.046,E2 -7667.046} C_VEL
LIN {X 0,Y 471.601,Z 453.605,A -85,B 0,C 180,E1 -7667.676,E2 -7667.676} C_VEL
LIN {X 0,Y 471.567,Z 448.773,A -85,B 0,C 180,E1 -7667.863,E2 -7667.863} C_VEL
LIN {X 0,Y 468.688,Z 434.641,A -85,B 0,C 180,E1 -7668.403,E2 -7668.403} C_VEL
LIN {X 0,Y 466.969,Z 427.179,A -85,B 0,C 180,E1 -7668.636,E2 -7668.636} C_VEL
LIN {X 0,Y 467.083,Z 422.04,A -85,B 0,C 180,E1 -7671.169,E2 -7671.169} C_VEL
LIN {X 0,Y 467.177,Z 416.463,A -85,B 0,C 180,E1 -7673.965,E2 -7673.965} C_VEL
LIN {X 0,Y 467.351,Z 410.905,A -85,B 0,C 180,E1 -7676.817,E2 -7676.817} C_VEL
LIN {X 0,Y 467.521,Z 405.345,A -85,B 0,C 180,E1 -7679.74,E2 -7679.74} C_VEL
LIN {X 0,Y 467.777,Z 399.802,A -85,B 0,C 180,E1 -7682.743,E2 -7682.743} C_VEL
